	120:
	// Set Parameters to read the Micro Controller (MC1) 3300mv Nominal Voltage INPUT of the EK1914.
		fbCoERead.nSubIndex := 16#01;
		fbCoERead.nIndex 	:= 16#FA81;
		fbCoERead.pDstBuf	:= 	ADR(wEK1914_MC1_3300mV);
		fbCoERead.cbBufLen	:= 	SIZEOF(wEK1914_MC1_3300mV);
		fbCoERead.bExecute	:= TRUE;
		iState := iState + 10;
		
	130:// Evaluate read of the Micro Controller (MC1) 3300mv Nominal Voltage INPUT of the EK1914.		
		IF NOT fbCoERead.bBusy THEN
			q_stEK1914_Diag.lrMC1_3300mV  :=  WORD_TO_LREAL(wEK1914_MC1_3300mV);
			fbCoERead.bExecute	:= FALSE;
			q_sErrorDescription := 'No Error';
			iState := iState + 10;
		ELSIF fbCoERead.bError THEN
			q_sErrorDescription := 'EK1914 MC1 3.3v Input - Read Error';
		END_IF							

	140:
	// Set Parameters to read the Micro Controller (MC2) 3300mv Nominal Voltage INPUT of the EK1914.
		fbCoERead.nSubIndex := 16#02;
		fbCoERead.nIndex 	:= 16#FA81;
		fbCoERead.pDstBuf	:= 	ADR(wEK1914_MC2_3300mV);
		fbCoERead.cbBufLen	:= 	SIZEOF(wEK1914_MC2_3300mV);
		fbCoERead.bExecute	:= TRUE;
		iState := iState + 10;
		
	150:// Evaluate read of the Micro Controller (MC2) 3300mv Nominal Voltage INPUT of the EK1914.		
		IF NOT fbCoERead.bBusy THEN
			q_stEK1914_Diag.lrMC2_3300mV  :=  WORD_TO_LREAL(wEK1914_MC2_3300mV);
			fbCoERead.bExecute	:= FALSE;
			q_sErrorDescription := 'No Error';
			iState := iState + 10;
		ELSIF fbCoERead.bError THEN
			q_sErrorDescription := 'EK1914 MC2 3.3v Input - Read Error';
		END_IF		
	
	160:// Set Parameters to read Standard Output Active/Inactive of the EK1914.
		(* Standard outputs can be used to directly Enable/Disable a TwinSAFE output
	   		if this feature is ACTIVE (Not to Turn it ON/OFF, Allow it or not to turn ON!!! *)
		fbCoERead.nSubIndex := 16#01;
		fbCoERead.nIndex 	:= 16#8000;
		fbCoERead.pDstBuf	:= 	ADR(bEK1914_StandardOuts);
		fbCoERead.cbBufLen	:= 	SIZEOF(bEK1914_StandardOuts);
		fbCoERead.bExecute	:= TRUE;
		iState := iState + 10;
	
	170:// Evaluate read of Standard Output Active/Inactive of the EK1914.
		IF NOT fbCoERead.bBusy THEN								
			q_stEK1914_Diag.xStandardOutputActive  :=  bEK1914_StandardOuts.0 ;
			fbCoERead.bExecute	:= FALSE;
			q_sErrorDescription := 'No Error';
			iState := iState + 10;
		ELSIF fbCoERead.bError THEN
			q_sErrorDescription := 'EK1914 Standard Outputs Active - Read Error';
		END_IF							

	180://Set Parameters to read Test Pulses Active/Inactive of the EK1914.
		(* Used to determine TwinSAFE output wiring is correct *)
		fbCoERead.nSubIndex := 16#03;
		fbCoERead.nIndex 	:= 16#8000;
		fbCoERead.pDstBuf	:= 	ADR(bEK1914_TestP);
		fbCoERead.cbBufLen	:= 	SIZEOF(bEK1914_TestP);
		fbCoERead.bExecute	:= TRUE;
		iState := iState + 10;
		
	190:// Evaluate read of Test Pulses Active/Inactive of the EK1914.
		IF NOT fbCoERead.bBusy THEN								
			q_stEK1914_Diag.xTestPulsesActive  :=  bEK1914_TestP.0 ;
			fbCoERead.bExecute	:= FALSE;
			q_sErrorDescription := 'No Error';
			iState := iState + 10;
		ELSIF fbCoERead.bError THEN
			q_sErrorDescription := 'EK1914 Test Pulses Active/Inactive - Read Error';
		END_IF		

	200:// Set Parameters to read Output Error Acknowledge Active/Inactive of the EK1914.
		(* Used to reset TwinSAFE output errors instead of forcing a cycle power
			for a TwinSAFE output error. *)
		fbCoERead.nSubIndex := 16#04;
		fbCoERead.nIndex 	:= 16#8000;
		fbCoERead.pDstBuf	:= 	ADR(bEK1914_ErrAck);
		fbCoERead.cbBufLen	:= 	SIZEOF(bEK1914_ErrAck);
		fbCoERead.bExecute	:= TRUE;
		iState := iState + 10;
		
	210:// Evaluate read of Output Error Acknowledge Active/Inactive of the EK1914.	
		IF NOT fbCoERead.bBusy THEN								
			q_stEK1914_Diag.xOutputErrAckActive  :=  bEK1914_ErrAck.0 ;
			fbCoERead.bExecute	:= FALSE;
			q_sErrorDescription := 'No Error';
			iState := iState + 10;
		ELSIF fbCoERead.bError THEN
			q_sErrorDescription := 'EK1914 Output Error Acknowledge Active/Inactive - Read Error';
		END_IF						
		
	220:// Set Parameters to read Sensor Tests Active/Inactive Channel 1 of the EK1914.
		fbCoERead.nSubIndex := 1;
		fbCoERead.nIndex 	:= 16#8001;
		fbCoERead.pDstBuf	:= 	ADR(iEK1914_STActive1);
		fbCoERead.cbBufLen	:= 	SIZEOF(iEK1914_STActive1);
		fbCoERead.bExecute	:= TRUE;
		iState := iState + 10;
	
	230:// Evaluate read of	Sensor Tests Active/Inactive Channel 1 of the EK1914.
		IF NOT fbCoERead.bBusy THEN								
			IF NOT iEK1914_STActive1 THEN
				q_stEK1914_Diag.xSensorTestActive1 := FALSE;
			ELSIF iEK1914_STActive1 THEN
				q_stEK1914_Diag.xSensorTestActive1 := TRUE;
			END_IF
			fbCoERead.bExecute	:= FALSE;
			q_sErrorDescription := 'No Error';
			iState := iState + 10;
		ELSIF fbCoERead.bError THEN
			q_sErrorDescription := 'EK1914 Sensor Tests Active/Inactive Channel 1 - Read Error';
		END_IF						
		
	240:// Set Parameters to read Sensor Tests Active/Inactive Channel 2 of the EK1914.
		fbCoERead.nSubIndex := 2;
		fbCoERead.nIndex 	:= 16#8001;
		fbCoERead.pDstBuf	:= 	ADR(iEK1914_STActive2);
		fbCoERead.cbBufLen	:= 	SIZEOF(iEK1914_STActive2);
		fbCoERead.bExecute	:= TRUE;
		iState := iState + 10;
		
	250:// Evaluate read of	Sensor Tests Active/Inactive Channel 1 of the EK1914.
		IF NOT fbCoERead.bBusy THEN								
			IF NOT iEK1914_STActive2 THEN
				q_stEK1914_Diag.xSensorTestActive2 := FALSE;
			ELSIF iEK1914_STActive2 THEN
				q_stEK1914_Diag.xSensorTestActive2 := TRUE;
			END_IF
			fbCoERead.bExecute	:= FALSE;
			q_sErrorDescription := 'No Error';
			iState := iState + 10;
		ELSIF fbCoERead.bError THEN
			q_sErrorDescription := 'EK1914 Sensor Tests Active/Inactive Channel 2 - Read Error';
		END_IF						
		
	260:// Set Parameters to read the Logic setting of Channels 1 and 2 of the EK1914.
		fbCoERead.nSubIndex := 1;
		fbCoERead.nIndex 	:= 16#8002;
		fbCoERead.pDstBuf	:= 	ADR(bEK1914_Logic1_2);
		fbCoERead.cbBufLen	:= 	SIZEOF(bEK1914_Logic1_2);
		fbCoERead.bExecute	:= TRUE;
		iState := iState + 10;
		
	270:// Evaluate read of the Logic setting of Channels 1 and 2 of the EK1914.
		IF NOT fbCoERead.bBusy THEN								
			IF  bEK1914_Logic1_2  = 0  THEN
				q_stEK1914_Diag.sLogicMode_Ch1Ch2 := 'Single Channel Logic.' ;
			ELSIF  bEK1914_Logic1_2  =  1  THEN
				q_stEK1914_Diag.sLogicMode_Ch1Ch2 := 'Asynchronous Repetitive OSSD, Sensor Test Must Be Disabled!' ;
			ELSIF  bEK1914_Logic1_2  =  2  THEN
				q_stEK1914_Diag.sLogicMode_Ch1Ch2 := 'Any Pulse Repetitive OSSD, Sensor Test Must Be Disabled!' ;
			ELSIF  bEK1914_Logic1_2  =  3  THEN
				q_stEK1914_Diag.sLogicMode_Ch1Ch2 := 'Short Cut, No Module Fault.' ;
			ELSE
				q_stEK1914_Diag.sLogicMode_Ch1Ch2 := 'Invalid Logic CH1 and CH2' ;
			END_IF ;		
			fbCoERead.bExecute	:= FALSE;
			q_sErrorDescription := 'No Error';
			iState := iState + 10;
		ELSIF fbCoERead.bError THEN
			q_sErrorDescription := 'EK1914 Logic setting of Channels 1 and 2 - Read Error';
		END_IF						
	
	
(**************************************ALARMS**************************************)
(**************************************ALARMS**************************************)
(**************************************ALARMS**************************************)
	280:// Set Parameters to read the Sensor Test state of the EK1914.	
		fbCoERead.nSubIndex := 16#0A;
		fbCoERead.nIndex 	:= 16#800E;
		fbCoERead.pDstBuf	:= 	ADR(wEK1914_SenT);
		fbCoERead.cbBufLen	:= 	SIZEOF(wEK1914_SenT);
		fbCoERead.bExecute	:= TRUE;
		iState := iState + 10;

	290:// Evaluate read of the Sensor Test state of the EK1914.
		IF NOT fbCoERead.bBusy THEN									
		(* These errors may only be present temporarily so they need to be latched and then cleared
			to be properly noted by the operator. *)
			IF wEK1914_SenT.0 OR wEK1914_SenT.1 THEN
				q_stEK1914_Diag.xSensorTest1_Error 	:= 	wEK1914_SenT.0;
				q_stEK1914_Diag.xSensorTest2_Error 	:= 	wEK1914_SenT.1;
			ELSIF i_xLatchedMessageReset THEN
				q_stEK1914_Diag.xSensorTest1_Error	:= FALSE;
				q_stEK1914_Diag.xSensorTest2_Error	:= FALSE;
			END_IF		
			fbCoERead.bExecute	:= FALSE;
			q_sErrorDescription := 'No Error';
			iState := iState + 10;
		ELSIF fbCoERead.bError THEN
			q_sErrorDescription := 'EK1914 Sensor Test - Read Error';
		END_IF						

	300:// Set Parameters to read the Two-Channel Evaluation Error - Diagnostic object 800E:0B
		(* The two channels contradict each other (not same value). *)
		fbCoERead.nSubIndex := 16#0B;
		fbCoERead.nIndex 	:= 16#800E;
		fbCoERead.pDstBuf	:= 	ADR(wEK1914_2CHEval);
		fbCoERead.cbBufLen	:= 	SIZEOF(wEK1914_2CHEval);
		fbCoERead.bExecute	:= TRUE;
		iState := iState + 10;

	310:// Evalutate read ofthe Two-Channel Evaluation Error - Diagnostic object 800E:0B
		(* The two channels contradict each other (not same value). *)
		IF NOT fbCoERead.bBusy THEN								
		(* These errors may only be present temporarily so they need to be latched and then cleared
			to be properly noted by the operator. *)
			IF wEK1914_2CHEval.0 OR wEK1914_2CHEval.1 THEN
				q_stEK1914_Diag.x2ChanEvalError_Pair1	 :=  wEK1914_2CHEval.0;
			ELSIF i_xLatchedMessageReset THEN
				q_stEK1914_Diag.x2ChanEvalError_Pair1	:= FALSE;
			END_IF	
			fbCoERead.bExecute	:= FALSE;
			q_sErrorDescription := 'No Error';
			iState := iState + 10;
		ELSIF fbCoERead.bError THEN
			q_sErrorDescription := 'EK1914 Two-Channel Evaluation Error - Read Error';
		END_IF						
		
	320:// Set Parameters to read Error In Safety Mat Operating Mode: Input Pair Disagree - Diagnostic object 800E:0C
		(* Input pairs not in the same state (not same value). *)
		fbCoERead.nSubIndex := 16#0C;
		fbCoERead.nIndex 	:= 16#800E;
		fbCoERead.pDstBuf	:= 	ADR(wEK1914_SMiPair);
		fbCoERead.cbBufLen	:= 	SIZEOF(wEK1914_SMiPair);
		fbCoERead.bExecute	:= TRUE;
		iState := iState + 10;
		
	330:// Evaluate read of Error In Safety Mat Operating Mode: Input Pair Disagree - Diagnostic object 800E:0C 
		(* Input pairs not in the same state (not same value). *)
		IF NOT fbCoERead.bBusy THEN								
		(* These errors may only be present temporarily so they need to be latched and then cleared
			to be properly noted by the operator. *)
			IF (wEK1914_SMiPair.0 AND wEK1914_SMiPair.1) THEN
				q_stEK1914_Diag.xSafeMatError_Pair1	 :=  (wEK1914_SMiPair.0  AND  wEK1914_SMiPair.1);
			ELSIF i_xLatchedMessageReset THEN
				q_stEK1914_Diag.xSafeMatError_Pair1	:= FALSE;
			END_IF	
			fbCoERead.bExecute	:= FALSE;
			q_sErrorDescription := 'No Error';
			iState := iState + 10;
		ELSIF fbCoERead.bError THEN
			q_sErrorDescription := 'EK1914 Error In Safety Mat: Input Pair Disagree - Read Error';
		END_IF						
		
	340:// Set Parameters to read Error In Safety Mat Operating Mode: External Supply (No test pulses) - Diagnostic object 800E:0D
		(* External supply detected (Input channel not getting test pulses). *)
		fbCoERead.nSubIndex := 16#0D;
		fbCoERead.nIndex 	:= 16#800E;
		fbCoERead.pDstBuf	:= 	ADR(wEK1914_SMExtSupply);
		fbCoERead.cbBufLen	:= 	SIZEOF(wEK1914_SMExtSupply);
		fbCoERead.bExecute	:= TRUE;
		iState := iState + 10;
		
	350:// Evaluate read Error In Safety Mat Operating Mode: External Supply (No test pulses) - Diagnostic object 800E:0D
		(* External supply detected (Input channel not getting test pulses). *)
		IF NOT fbCoERead.bBusy THEN								
		(* These errors may only be present temporarily so they need to be latched and then cleared
			to be properly noted by the operator. *)
			IF wEK1914_SMExtSupply > 0  THEN
				q_stEK1914_Diag.xSafeMatExternalSupplyErrorCh1  := 	wEK1914_SMExtSupply.0;
				q_stEK1914_Diag.xSafeMatExternalSupplyErrorCh2  := 	wEK1914_SMExtSupply.2;
			ELSIF i_xLatchedMessageReset THEN
				q_stEK1914_Diag.xSafeMatExternalSupplyErrorCh1	:= FALSE;
				q_stEK1914_Diag.xSafeMatExternalSupplyErrorCh2	:= FALSE;
			END_IF
			fbCoERead.bExecute	:= FALSE;
			q_sErrorDescription := 'No Error';
			iState := iState + 10;
		ELSIF fbCoERead.bError THEN
			q_sErrorDescription := 'EK1914 Error In Safety Mat: External Supply - Read Error';
		END_IF						
		
	360:// Set Parameters to read Error At The Output MC1 of the EK1914.
		(* External supply or cross-circuit Error Open Load, Current Below 20mA, OR Current Above Maximum Value OF 500mA. *)
		fbCoERead.nSubIndex := 16#0E;
		fbCoERead.nIndex 	:= 16#800E;
		fbCoERead.pDstBuf	:= 	ADR(wEK1914_OutErrMC1);
		fbCoERead.cbBufLen	:= 	SIZEOF(wEK1914_OutErrMC1);
		fbCoERead.bExecute	:= TRUE;
		iState := iState + 10;
		
	370:// Evaluate read Error At The Output MC1 of the EK1914.
		(* External supply or cross-circuit Error Open Load, Current Below 20mA, OR Current Above Maximum Value OF 500mA. *)	
		IF NOT fbCoERead.bBusy THEN														
		(* These errors may only be present temporarily so they need to be latched and then cleared
			to be properly noted by the operator. *)
			IF wEK1914_OutErrMC1 = 5 THEN
				q_stEK1914_Diag.xCrossCircuitError1_MC1 := TRUE;
				q_stEK1914_Diag.sOutputErrorDescription_MC1 := 'Cross-circuit output 1 and output 2.';
			ELSIF wEK1914_OutErrMC1 = 6 THEN
				q_stEK1914_Diag.xCrossCircuitError2_MC1 := TRUE;
				q_stEK1914_Diag.sOutputErrorDescription_MC1 := 'Cross-circuit output 1 and output 2.';
			ELSIF wEK1914_OutErrMC1 = 10 THEN
				q_stEK1914_Diag.xOverVoltage_MC1 := TRUE;
				q_stEK1914_Diag.sOutputErrorDescription_MC1 := 'Overvoltage.';
			ELSIF wEK1914_OutErrMC1 = 11 THEN
				q_stEK1914_Diag.xUnderVoltage_MC1 := TRUE;
				q_stEK1914_Diag.sOutputErrorDescription_MC1 := 'Undervoltage.';
			ELSIF (wEK1914_OutErrMC1 >= 21) AND (wEK1914_OutErrMC1 <= 27) THEN
				q_stEK1914_Diag.xFieldVoltageError_MC1 := TRUE;
				q_stEK1914_Diag.sOutputErrorDescription_MC1 := 'Error when testing the field voltage switches.';
			ELSIF (wEK1914_OutErrMC1 >= 30) AND (wEK1914_OutErrMC1 <= 33) THEN
				q_stEK1914_Diag.xStartupOutCircuitError_MC1 := TRUE;
				q_stEK1914_Diag.sOutputErrorDescription_MC1 := 'Start-up of the output circuit failed.';
			ELSIF wEK1914_OutErrMC1 = 101 THEN
				q_stEK1914_Diag.xExternalSupply0vError1_MC1 := TRUE;
				q_stEK1914_Diag.sOutputErrorDescription_MC1 := 'External supply 0v output 1, detected with set output.';
			ELSIF wEK1914_OutErrMC1 = 102 THEN
				q_stEK1914_Diag.xExternalSupply24vError1_MC1 := TRUE;
				q_stEK1914_Diag.sOutputErrorDescription_MC1 := 'External supply 24v output 1.';
			ELSIF wEK1914_OutErrMC1 = 103 THEN
				q_stEK1914_Diag.xExternalSupply0vError2_MC1 := TRUE;
				q_stEK1914_Diag.sOutputErrorDescription_MC1 := 'External supply 0v output 2, detected with set output.';
			ELSIF wEK1914_OutErrMC1 = 104 THEN
				q_stEK1914_Diag.xExternalSupply24vError2_MC1 := TRUE;
				q_stEK1914_Diag.sOutputErrorDescription_MC1 := 'External supply 24v output 2.';
			ELSE
				q_stEK1914_Diag.xExternalSupply24vError2_MC1 := FALSE;
				q_stEK1914_Diag.sOutputErrorDescription_MC1 := 'No Error.';
			END_IF
			fbCoERead.bExecute	:= FALSE;
			q_sErrorDescription := 'No Error';
			iState := iState + 10;
		ELSIF fbCoERead.bError THEN
			q_sErrorDescription := 'EK1914 Error At The Output (MC1) - Read Error';
		END_IF		
		
	380:// Set Parameters to read Error At The Output MC2 of the EK1914.
		(* External supply or cross-circuit Error Open Load, Current Below 20mA, OR Current Above Maximum Value OF 500mA. *)
		fbCoERead.nSubIndex := 16#0F;
		fbCoERead.nIndex 	:= 16#800E;
		fbCoERead.pDstBuf	:= 	ADR(wEK1914_OutErrMC2);
		fbCoERead.cbBufLen	:= 	SIZEOF(wEK1914_OutErrMC2);
		fbCoERead.bExecute	:= TRUE;
		iState := iState + 10;
	
	390:// Evaluate read of Error At The Output MC2 of the EK1914.
		(* External supply or cross-circuit Error Open Load, Current Below 20mA, OR Current Above Maximum Value OF 500mA. *)
		IF NOT fbCoERead.bBusy THEN	
		(* These errors may only be present temporarily so they need to be latched and then cleared
			to be properly noted by the operator. *)
			IF wEK1914_OutErrMC2 = 5 THEN
				q_stEK1914_Diag.xCrossCircuitError1_MC2 := TRUE;
				q_stEK1914_Diag.sOutputErrorDescription_MC2 := 'Cross-circuit output 1 and output 2 MC2.';
			ELSIF wEK1914_OutErrMC2 = 6 THEN
				q_stEK1914_Diag.xCrossCircuitError2_MC2 := TRUE;
				q_stEK1914_Diag.sOutputErrorDescription_MC2 := 'Cross-circuit output 1 and output 2 MC2.';
			ELSIF wEK1914_OutErrMC2 = 10 THEN
				q_stEK1914_Diag.xOverVoltage_MC2 := TRUE;
				q_stEK1914_Diag.sOutputErrorDescription_MC2 := 'Overvoltage MC2.';
			ELSIF wEK1914_OutErrMC2 = 11 THEN
				q_stEK1914_Diag.xUnderVoltage_MC2 := TRUE;
				q_stEK1914_Diag.sOutputErrorDescription_MC2 := 'Undervoltage.';
			ELSIF (wEK1914_OutErrMC2 >= 21) AND (wEK1914_OutErrMC2 <= 27) THEN
				q_stEK1914_Diag.xFieldVoltageError_MC2 := TRUE;
				q_stEK1914_Diag.sOutputErrorDescription_MC2 := 'Error when testing the field voltage switches MC2.';
			ELSIF (wEK1914_OutErrMC2 >= 30) AND (wEK1914_OutErrMC2 <= 33) THEN
				q_stEK1914_Diag.xStartupOutCircuitError_MC2 := TRUE;
				q_stEK1914_Diag.sOutputErrorDescription_MC2 := 'Start-up of the output circuit failed MC2.';
			ELSIF wEK1914_OutErrMC2 = 101 THEN
				q_stEK1914_Diag.xExternalSupply0vError1_MC2 := TRUE;
				q_stEK1914_Diag.sOutputErrorDescription_MC2 := 'External supply 0v output 1, detected with set output MC2.';
			ELSIF wEK1914_OutErrMC2 = 102 THEN
				q_stEK1914_Diag.xExternalSupply24vError1_MC2 := TRUE;
				q_stEK1914_Diag.sOutputErrorDescription_MC2 := 'External supply 24v output 1 MC2.';
			ELSIF wEK1914_OutErrMC2 = 103 THEN
				q_stEK1914_Diag.xExternalSupply0vError2_MC2 := TRUE;
				q_stEK1914_Diag.sOutputErrorDescription_MC2 := 'External supply 0v output 2, detected with set output MC2.';
			ELSIF wEK1914_OutErrMC2 = 104 THEN
				q_stEK1914_Diag.xExternalSupply24vError2_MC2 := TRUE;
				q_stEK1914_Diag.sOutputErrorDescription_MC2 := 'External supply 24v output 2 MC2.';
			ELSE
				q_stEK1914_Diag.xExternalSupply24vError2_MC2 := FALSE;
				q_stEK1914_Diag.sOutputErrorDescription_MC2 := 'No Error.';
			END_IF
			fbCoERead.bExecute	:= FALSE;
			q_sErrorDescription := 'No Error';
			iState := iState + 10;
		ELSIF fbCoERead.bError THEN
			q_sErrorDescription := 'EK1914 Error At The Output (MC2) - Read Error';
		END_IF								

	400:// Set Parameters to read Connection State of the EK1914.
		fbCoERead.nSubIndex := 1;
		fbCoERead.nIndex 	:= 16#A000;
		fbCoERead.pDstBuf	:= 	ADR(iEK1914_ConnectionState);
		fbCoERead.cbBufLen	:= 	SIZEOF(iEK1914_ConnectionState);
		fbCoERead.bExecute	:= TRUE;
		iState := iState + 10;
		
	410:// Evaluate read of the Connection State of the EK1914.
		IF NOT fbCoERead.bBusy THEN								
			IF iEK1914_ConnectionState = 100 THEN
				q_stEK1914_Diag.sConnectionState := 'Reset State';
			ELSIF iEK1914_ConnectionState = 101 THEN
				q_stEK1914_Diag.sConnectionState := 'Session State';
			ELSIF iEK1914_ConnectionState = 102 THEN
				q_stEK1914_Diag.sConnectionState := 'Connection State';
			ELSIF iEK1914_ConnectionState = 103 THEN
				q_stEK1914_Diag.sConnectionState := 'Parameter State';
			ELSIF iEK1914_ConnectionState = 104 THEN
				q_stEK1914_Diag.sConnectionState := 'Data State';
			ELSIF iEK1914_ConnectionState = 105 THEN
				q_stEK1914_Diag.sConnectionState := 'Failsafe State';
			ELSE
				q_stEK1914_Diag.sConnectionState := 'Undefined State';
			END_IF
			fbCoERead.bExecute	:= FALSE;
			q_sErrorDescription := 'No Error';
			iState := 0;
		ELSIF fbCoERead.bError THEN
			q_sErrorDescription := 'EK1914 Connection State - Read Error';
		END_IF	
END_CASE

// FB_EcCoESdoRead for all CoE reads.
fbCoERead(
	sNetId:= i_sNetId, 
	nSlaveAddr:= i_nSlaveAddr, 
	nSubIndex:= , 
	nIndex:= , 
	pDstBuf:= , 
	cbBufLen:= , 
	bExecute:= , 
	tTimeout:= T#2S, 
	bBusy=> , 
	bError=> q_xError, 
	nErrId=> q_udiErrorID);

// If any of above errors exist set q_stEK1914_Diag.xEK1914Error TRUE.
IF NOT q_stEK1914_Diag.xSensorTest1_Error OR
		q_stEK1914_Diag.xSensorTest2_Error OR
		q_stEK1914_Diag.x2ChanEvalError_Pair1 OR
		q_stEK1914_Diag.xSafeMatError_Pair1 OR
		q_stEK1914_Diag.xSafeMatExternalSupplyErrorCh1 OR
		q_stEK1914_Diag.xSafeMatExternalSupplyErrorCh2 OR 
		q_stEK1914_Diag.xCrossCircuitError1_MC1 OR 
		q_stEK1914_Diag.xCrossCircuitError2_MC1 OR 
		q_stEK1914_Diag.xOverVoltage_MC1 OR 
		q_stEK1914_Diag.xUnderVoltage_MC1 OR
		q_stEK1914_Diag.xFieldVoltageError_MC1 OR 
		q_stEK1914_Diag.xStartupOutCircuitError_MC1 OR 
		q_stEK1914_Diag.xExternalSupply0vError1_MC1 OR 
		q_stEK1914_Diag.xExternalSupply24vError1_MC1 OR 
		q_stEK1914_Diag.xExternalSupply0vError2_MC1 OR 
		q_stEK1914_Diag.xExternalSupply24vError2_MC1 OR
		q_stEK1914_Diag.xCrossCircuitError1_MC2 OR 
		q_stEK1914_Diag.xCrossCircuitError2_MC2 OR 
		q_stEK1914_Diag.xOverVoltage_MC2 OR 
		q_stEK1914_Diag.xUnderVoltage_MC2 OR
		q_stEK1914_Diag.xFieldVoltageError_MC2 OR 
		q_stEK1914_Diag.xStartupOutCircuitError_MC2 OR 
		q_stEK1914_Diag.xExternalSupply0vError1_MC2 OR 
		q_stEK1914_Diag.xExternalSupply24vError1_MC2 OR 
		q_stEK1914_Diag.xExternalSupply0vError2_MC2 OR 
		q_stEK1914_Diag.xExternalSupply24vError2_MC2 THEN
			q_stEK1914_Diag.xEK1914Error := FALSE;
ELSIF q_stEK1914_Diag.xSensorTest1_Error OR
		q_stEK1914_Diag.xSensorTest2_Error OR
		q_stEK1914_Diag.x2ChanEvalError_Pair1 OR
		q_stEK1914_Diag.xSafeMatError_Pair1 OR
		q_stEK1914_Diag.xSafeMatExternalSupplyErrorCh1 OR
		q_stEK1914_Diag.xSafeMatExternalSupplyErrorCh2 OR 
		q_stEK1914_Diag.xCrossCircuitError1_MC1 OR 
		q_stEK1914_Diag.xCrossCircuitError2_MC1 OR 
		q_stEK1914_Diag.xOverVoltage_MC1 OR 
		q_stEK1914_Diag.xUnderVoltage_MC1 OR
		q_stEK1914_Diag.xFieldVoltageError_MC1 OR 
		q_stEK1914_Diag.xStartupOutCircuitError_MC1 OR 
		q_stEK1914_Diag.xExternalSupply0vError1_MC1 OR 
		q_stEK1914_Diag.xExternalSupply24vError1_MC1 OR 
		q_stEK1914_Diag.xExternalSupply0vError2_MC1 OR 
		q_stEK1914_Diag.xExternalSupply24vError2_MC1 OR
		q_stEK1914_Diag.xCrossCircuitError1_MC2 OR 
		q_stEK1914_Diag.xCrossCircuitError2_MC2 OR 
		q_stEK1914_Diag.xOverVoltage_MC2 OR 
		q_stEK1914_Diag.xUnderVoltage_MC2 OR
		q_stEK1914_Diag.xFieldVoltageError_MC2 OR 
		q_stEK1914_Diag.xStartupOutCircuitError_MC2 OR 
		q_stEK1914_Diag.xExternalSupply0vError1_MC2 OR 
		q_stEK1914_Diag.xExternalSupply24vError1_MC2 OR 
		q_stEK1914_Diag.xExternalSupply0vError2_MC2 OR 
		q_stEK1914_Diag.xExternalSupply24vError2_MC2 THEN
			q_stEK1914_Diag.xEK1914Error := TRUE;
END_IF

END_FUNCTION_BLOCK

// POUs/HardwareFBs/FB_EL69xxDiagnostics
(*=====================================================================
Beckhoff Automation LLC
Copyright 2015 All Rights Reserved
=======================================================================
Description: 
This Program has been supplied by Beckhoff Automation As-Is and is intended only as an example implementation. 
Functionality is not guaranteed. 
This Function Block reads all status and error information known at time of creation of the EL69xx.
---------------------------------------------------------------------------------------------------------------
History:
Date		Version			Author							Comment
---------------------------------------------------------------------------------------------------------------
07.08.15	0.10		Jason Erickson				Initial Library Creation.
07.20.15	0.11		Jason Ericskon				Added CoE Read for TwinSAFE Connection State.
08.28.15	0.20		Jason Erickson				Code optimization to eliminate timed data reads.
09.18.15	0.2.1		Jason Erickson				Added new error codes 0x6000 - 0x6002 and Connection Status to the AX5805.
09.24.15	0.2.2		Jason Erickson				Corrected inability to update CASE in FB_EL1904Diagnostics and FB_EL2904Diagnostics.
10.30.15	0.2.3		Jason Erickson				Modified Diagnostic Structure names for ease of use.
*)
FUNCTION_BLOCK FB_EL69xxDiagnostics
VAR_INPUT
// EtherCAT Master Device Net ID.
	i_sNetId: STRING;
// Slave Address of the EL69xx.
	i_nSlaveAddr: UINT;
// Input to reset Latched TwinSAFE Error Messages.
	i_xLatchedMessageReset: BOOL;
END_VAR
VAR_OUTPUT
// Structure to hold all EL69xx output information.
	q_stEL69xx_Diag: ST_EL69xx_DIAGNOSTICS;
// Internal function block errors.
	q_xError: BOOL;
	q_udiErrorID: UDINT;
	q_sErrorDescription: STRING;
END_VAR
VAR
// Case Statement.
	iState: INT;
// FB_EcCoESdoRead for all CoE reads.
	fbCoERead: FB_EcCoESdoRead;
// Variable to hold data for evaluation, Micro Controller (MC1) 3.3v Nominal Voltage(mV) INPUT of the EL69xx.
	wEL69xx_MC1_3300mV: WORD;
// Variable to hold data for evaluation, Micro Controller (MC2) 3.3v Nominal Voltage(mV) INPUT of the EL69xx.
	wEL69xx_MC2_3300mV: WORD;
// Variable to hold data for evaluation, Temperature and Voltage Errors of the EL69xx.
	(* There are two temperature sensors inside each Microcontroller. *)
	wEL69xx_Error: WORD;
END_VAR

CASE iState OF
	0:
	// Set Parameters to read Serial Number of the EL69xx.	
		fbCoERead.nSubIndex := 16#02;
		fbCoERead.nIndex 	:= 16#F980;
		fbCoERead.pDstBuf	:= 	ADR(q_stEL69xx_Diag.dwSerialNumber);
		fbCoERead.cbBufLen	:= 	SIZEOF(q_stEL69xx_Diag.dwSerialNumber);
		fbCoERead.bExecute	:= TRUE;
		iState := iState + 10;
		
	10:// Evaluate read of the Serial Number of the EL69xx.
		IF NOT fbCoERead.bBusy THEN
			fbCoERead.bExecute	:= FALSE;
			q_sErrorDescription := 'No Error';
			iState := iState + 10;
		ELSIF fbCoERead.bError THEN
			q_sErrorDescription := 'EL69xx Serial Number - Read Error';
		END_IF
	
	20:// Set Parameters to read DIP Switch setting out of the EL69xx.
		fbCoERead.nSubIndex := 16#01;
		fbCoERead.nIndex 	:= 16#F980;
		fbCoERead.pDstBuf	:= 	ADR(q_stEL69xx_Diag.wDipSwitch);
		fbCoERead.cbBufLen	:= 	SIZEOF(q_stEL69xx_Diag.wDipSwitch);
		fbCoERead.bExecute	:= TRUE;
		iState := iState + 10;
		
	30:// Evaluate read of the DIP Switch setting of the EL69xx.
		IF NOT fbCoERead.bBusy THEN
			fbCoERead.bExecute	:= FALSE;
			q_sErrorDescription := 'No Error';
			iState := iState + 10;
		ELSIF fbCoERead.bError THEN
			q_sErrorDescription := 'EL69xx DIP Switch - Read Error';
		END_IF	
	
	40:// Set Parameters to read Hardware Version of the EL69xx.
		fbCoERead.nSubIndex := 0;
		fbCoERead.nIndex 	:= 16#1009;
		fbCoERead.pDstBuf	:= 	ADR(q_stEL69xx_Diag.sHwVersion);
		fbCoERead.cbBufLen	:= 	SIZEOF(q_stEL69xx_Diag.sHwVersion);
		fbCoERead.bExecute	:= TRUE;
		iState := iState + 10;
	
	50:// Evaluate read of Hardware Version of the EL69xx.
		IF NOT fbCoERead.bBusy THEN
			fbCoERead.bExecute	:= FALSE;
			q_sErrorDescription := 'No Error';
			iState := iState + 10;
		ELSIF fbCoERead.bError THEN
			q_sErrorDescription := 'EL69xx Hardware Version - Read Error';
		END_IF	

	60:// Set Parameters to read Software Version (firmware) of the EL69xx.
		fbCoERead.nSubIndex := 0;
		fbCoERead.nIndex 	:= 16#100A;
		fbCoERead.pDstBuf	:= 	ADR(q_stEL69xx_Diag.sFwVersion);
		fbCoERead.cbBufLen	:= 	SIZEOF(q_stEL69xx_Diag.sFwVersion);
		fbCoERead.bExecute	:= TRUE;
		iState := iState + 10;
	
	70:// Evaluate read of Software Version (firmware) of the EL69xx.
		IF NOT fbCoERead.bBusy THEN
			fbCoERead.bExecute	:= FALSE;
			q_sErrorDescription := 'No Error';
			iState := iState + 10;
		ELSIF fbCoERead.bError THEN
			q_sErrorDescription := 'EL69xx Software Version - Read Error';
		END_IF	

	80:// Set Parameters to read Micro Controller (MC1) Temperature in DegC of the EL69xx.
		fbCoERead.nSubIndex := 1;
		fbCoERead.nIndex 	:= 16#FA80;
		fbCoERead.pDstBuf	:= 	ADR(q_stEL69xx_Diag.wMC1Temp);
		fbCoERead.cbBufLen	:= 	SIZEOF(q_stEL69xx_Diag.wMC1Temp);
		fbCoERead.bExecute	:= TRUE;
		iState := iState + 10;
		
	90:// Evaluate read of Micro Controller (MC1) Temperature in DegC of the EL69xx.
		IF NOT fbCoERead.bBusy THEN
			fbCoERead.bExecute	:= FALSE;
			q_sErrorDescription := 'No Error';
			iState := iState + 10;
		ELSIF fbCoERead.bError THEN
			q_sErrorDescription := 'EL69xx MC1 Temp - Read Error';
		END_IF

	100:// Set Parameters to read Micro Controller (MC2) Temperature in DegC of the EL69xx.
		fbCoERead.nSubIndex := 2;
		fbCoERead.nIndex 	:= 16#FA80;
		fbCoERead.pDstBuf	:= 	ADR(q_stEL69xx_Diag.wMC2Temp);
		fbCoERead.cbBufLen	:= 	SIZEOF(q_stEL69xx_Diag.wMC2Temp);
		fbCoERead.bExecute	:= TRUE;
		iState := iState + 10;
		
	110:// Evaluate read of Micro Controller (MC2) Temperature in DegC of the EL69xx.
		IF NOT fbCoERead.bBusy THEN
			fbCoERead.bExecute	:= FALSE;
			q_sErrorDescription := 'No Error';
			iState := iState + 10;
		ELSIF fbCoERead.bError THEN
			q_sErrorDescription := 'EL69xx MC2 Temp - Read Error';
		END_IF

	120://Set Parameters to read Micro Controller (MC1) 3300mv Nominal Voltage INPUT of the EL69xx.
		fbCoERead.nSubIndex := 3;
		fbCoERead.nIndex 	:= 16#FA80;
		fbCoERead.pDstBuf	:= 	ADR(wEL69xx_MC1_3300mV);
		fbCoERead.cbBufLen	:= 	SIZEOF(wEL69xx_MC1_3300mV);
		fbCoERead.bExecute	:= TRUE;
		iState := iState + 10;
		
	130:// Evaluate read of Micro Controller (MC1) 3300mv Nominal Voltage INPUT of the EL69xx.
		IF NOT fbCoERead.bBusy THEN
			q_stEL69xx_Diag.lrMC1_3300mV  :=  WORD_TO_LREAL(wEL69xx_MC1_3300mV);
			fbCoERead.bExecute	:= FALSE;
			q_sErrorDescription := 'No Error';
			iState := iState + 10;
		ELSIF fbCoERead.bError THEN
			q_sErrorDescription := 'EL69xx MC1 3.3v Input - Read Error';
		END_IF

	140:// Set Parameters to read Micro Controller (MC2) 3300mv Nominal Voltage INPUT of the EL69xx.
		fbCoERead.nSubIndex := 4;
		fbCoERead.nIndex 	:= 16#FA80;
		fbCoERead.pDstBuf	:= 	ADR(wEL69xx_MC2_3300mV);
		fbCoERead.cbBufLen	:= 	SIZEOF(wEL69xx_MC2_3300mV);
		fbCoERead.bExecute	:= TRUE;
		iState := iState + 10;
		
	150:// Evaluate read of	Micro Controller (MC2) 3300mv Nominal Voltage INPUT of the EL69xx.
		IF NOT fbCoERead.bBusy THEN
			q_stEL69xx_Diag.lrMC2_3300mV  :=  WORD_TO_LREAL(wEL69xx_MC2_3300mV);
			fbCoERead.bExecute	:= FALSE;
			q_sErrorDescription := 'No Error';
			iState := iState + 10;
		ELSIF fbCoERead.bError THEN
			q_sErrorDescription := 'EL69xx MC2 3.3v Input Read - Error';
		END_IF
		
	160:// Set Parameters to read Temperature and Voltage Errors of the EL69xx.
		(* There are two temperature sensors inside each Microcontroller. *)
		fbCoERead.nSubIndex := 3;
		fbCoERead.nIndex 	:= 16#FA00;
		fbCoERead.pDstBuf	:= 	ADR(wEL69xx_Error);
		fbCoERead.cbBufLen	:= 	SIZEOF(wEL69xx_Error);
		fbCoERead.bExecute	:= TRUE;
		iState := iState + 10;
	
	170:// Evaluate read of	Temperature and Voltage Errors of the EL69xx.	
		(* There are two temperature sensors inside each Microcontroller. *)
		IF NOT fbCoERead.bBusy THEN
		(* These errors may only be present temporarily so they need to be latched and then cleared
			to be properly noted by the operator. *)
			IF wEL69xx_Error.2 OR wEL69xx_Error.8 THEN
				q_stEL69xx_Diag.xMaxTempError		:= 		(wEL69xx_Error = 5);
				q_stEL69xx_Diag.xMinTempError		:= 		(wEL69xx_Error = 6);
				q_stEL69xx_Diag.xTempDiffError	:= 		(wEL69xx_Error = 7);
				q_stEL69xx_Diag.xMaxVccMC1		:= 		(wEL69xx_Error = 257);
				q_stEL69xx_Diag.xMaxVccMC2		:= 		(wEL69xx_Error = 258);
				q_stEL69xx_Diag.xMinVccMC1		:= 		(wEL69xx_Error = 259);
				q_stEL69xx_Diag.xMinVccMC2		:= 		(wEL69xx_Error = 260);
			ELSIF i_xLatchedMessageReset THEN
				q_stEL69xx_Diag.xMaxTempError	:= FALSE;
				q_stEL69xx_Diag.xMinTempError	:= FALSE;
				q_stEL69xx_Diag.xTempDiffError:= FALSE;
				q_stEL69xx_Diag.xMaxVccMC1	:= FALSE;
				q_stEL69xx_Diag.xMaxVccMC2	:= FALSE;
				q_stEL69xx_Diag.xMinVccMC1	:= FALSE;
				q_stEL69xx_Diag.xMinVccMC2	:= FALSE;
			END_IF
			fbCoERead.bExecute	:= FALSE;
			q_sErrorDescription := 'No Error';
			iState := iState + 10;
		ELSIF fbCoERead.bError THEN
			q_sErrorDescription := 'EL69xx Temp and Voltage Error - Read Error';
		END_IF
		
	180:// Set Parameters to read Number of Safety Connections configured In The EL69xx.
		fbCoERead.nSubIndex := 0;
		fbCoERead.nIndex 	:= 16#2110;
		fbCoERead.pDstBuf	:= 	ADR(q_stEL69xx_Diag.bNumOfConnections);
		fbCoERead.cbBufLen	:= 	SIZEOF(q_stEL69xx_Diag.bNumOfConnections);
		fbCoERead.bExecute	:= TRUE;
		iState := iState + 10;
		
	190:// Evaluate read of Number of Safety Connections configured In The EL69xx.
		IF NOT fbCoERead.bBusy THEN
			fbCoERead.bExecute	:= FALSE;
			q_sErrorDescription := 'No Error';
			iState := iState + 10;
		ELSIF fbCoERead.bError THEN
			q_sErrorDescription := 'EL69xx Number of Safety Connections - Read Error';
		END_IF	

	200:// Set Parameters to read Number of Safety Groups Configured in the EL69xx.
		fbCoERead.nSubIndex := 0;
		fbCoERead.nIndex 	:= 16#2120;
		fbCoERead.pDstBuf	:= 	ADR(q_stEL69xx_Diag.bNumOfSafetyGroups);
		fbCoERead.cbBufLen	:= 	SIZEOF(q_stEL69xx_Diag.bNumOfSafetyGroups);
		fbCoERead.bExecute	:= TRUE;
		iState := iState + 10;
		
	210:// Evaluate read of Number of Safety Groups Configured in the EL69xx.	
		IF NOT fbCoERead.bBusy THEN
			fbCoERead.bExecute	:= FALSE;
			q_sErrorDescription := 'No Error';
			iState := iState + 10;
		ELSIF fbCoERead.bError THEN
			q_sErrorDescription := 'EL69xx Number of Safety Groups - Read Error';
		END_IF	
	
	220://Set Parameters to read Number of Safety Function Blocks Configured in the EL69xx.
		fbCoERead.nSubIndex := 0;
		fbCoERead.nIndex 	:= 16#2130;
		fbCoERead.pDstBuf	:= 	ADR(q_stEL69xx_Diag.bNumOfSafetyBlocks);
		fbCoERead.cbBufLen	:= 	SIZEOF(q_stEL69xx_Diag.bNumOfSafetyBlocks);
		fbCoERead.bExecute	:= TRUE;
		iState := iState + 10;
		
	230:// Evaluate read of	Number of Safety Function Blocks Configured in the EL69xx.
		IF NOT fbCoERead.bBusy THEN
			fbCoERead.bExecute	:= FALSE;
			q_sErrorDescription := 'No Error';
			iState := 0;
		ELSIF fbCoERead.bError THEN
			q_sErrorDescription := 'EL69xx Number of Safety Function Blocks Configured - Read Error';
		END_IF	
END_CASE

// FB_EcCoESdoRead for all CoE reads.
fbCoERead(
	sNetId:= i_sNetId, 
	nSlaveAddr:= i_nSlaveAddr, 
	nSubIndex:= , 
	nIndex:= , 
	pDstBuf:= , 
	cbBufLen:= , 
	bExecute:= , 
	tTimeout:= T#2S, 
	bBusy=> , 
	bError=> q_xError, 
	nErrId=> q_udiErrorID);

// If any of above errors exist set q_stEL69xx_Diag.xEL69xq_xError TRUE
IF NOT q_stEL69xx_Diag.xMaxTempError OR
	q_stEL69xx_Diag.xMinTempError OR
	q_stEL69xx_Diag.xMaxVccMC1 OR
	q_stEL69xx_Diag.xMaxVccMC2 OR
	q_stEL69xx_Diag.xMinVccMC1 OR
	q_stEL69xx_Diag.xMinVccMC2 OR
	q_stEL69xx_Diag.xTempDiffError THEN
		q_stEL69xx_Diag.xEL69xxError := FALSE;
ELSIF q_stEL69xx_Diag.xMaxTempError OR
	q_stEL69xx_Diag.xMinTempError OR
	q_stEL69xx_Diag.xMaxVccMC1 OR
	q_stEL69xx_Diag.xMaxVccMC2 OR
	q_stEL69xx_Diag.xMinVccMC1 OR
	q_stEL69xx_Diag.xMinVccMC2 OR
	q_stEL69xx_Diag.xTempDiffError THEN
		q_stEL69xx_Diag.xEL69xxError := TRUE;
END_IF

END_FUNCTION_BLOCK

// POUs/HardwareFBs/FB_EP1908Diagnostics
(*=====================================================================
Beckhoff Automation LLC
Copyright 2015 All Rights Reserved
=======================================================================
Description: 
This Program has been supplied by Beckhoff Automation As-Is and is intended only as an example implementation. 
Functionality is not guaranteed. 
This Function Block reads all status and error information known at time of creation of the EP1908.
---------------------------------------------------------------------------------------------------------------
History:
Date		Version			Author							Comment
---------------------------------------------------------------------------------------------------------------
07.08.15	0.10		Jason Erickson				Initial Library Creation.
07.20.15	0.11		Jason Ericskon				Added CoE Read for TwinSAFE Connection State.
08.28.15	0.20		Jason Erickson				Code optimization to eliminate timed data reads.
09.18.15	0.2.1		Jason Erickson				Added new error codes 0x6000 - 0x6002 and Connection Status to the AX5805.
09.24.15	0.2.2		Jason Erickson				Corrected inability to update CASE in FB_EL1904Diagnostics and FB_EL2904Diagnostics.
10.30.15	0.2.3		Jason Erickson				Modified Diagnostic Structure names for ease of use.
*)
FUNCTION_BLOCK FB_EP1908Diagnostics
VAR_INPUT
// EtherCAT Master Device Net ID.
	i_sNetId: STRING;
// Slave Address of the EP1908.		
	i_nSlaveAddr: UINT;
// Input to reset Latched TwinSAFE Error Messages.
	i_xLatchedMessageReset: BOOL;
END_VAR
VAR_OUTPUT
// Structure to hold all EP1908 output information.
	q_stEP1908_Diag: ST_EP1908_DIAGNOSTICS;
// Internal function block errors.
	q_xError: BOOL;
	q_nErrorID: UDINT;
	q_sErrorDescription: STRING;
END_VAR
VAR
// Case Statement.
	iState: INT;
// FB_EcCoESdoRead for all CoE reads.
	fbCoERead: FB_EcCoESdoRead;
// FB_EcCoESdoReadEx for all CoE EX reads.
	fbCoEReadEX: FB_EcCoESdoReadEx;
// Variable to hold data for evaluation, Micro Controller (MC1) 3.3v Nominal Voltage(mV) INPUT of the EP1908.	
	wEP1908_MC1_3300mV: WORD;
// Variable to hold data for evaluation, Micro Controller (MC2) 3.3v Nominal Voltage(mV) INPUT of the EP1908.	
	wEP1908_MC2_3300mV: WORD;
// Variable to hold data for evaluation, Operating Mode of the EP1908.
	wEP1908_OperMode: WORD;
// Variable to hold data for evaluation, Sensor Tests Active/Inactive of the EP1908.
	iSensorTestActive: INT;
// Variable to hold data for evaluation, Logic of the EP1908 Channels 1 and 2.
	bEP1908_Logic1_2: BYTE;
// Variable to hold data for evaluation, Logic of the EP1908 Channels 3 and 4.
	bEP1908_Logic3_4: BYTE;
// Variable to hold data for evaluation, Logic of the EP1908 Channels 5 and 6.
	bEP1908_Logic5_6: BYTE;
// Variable to hold data for evaluation, Logic of the EP1908 Channels 7 and 8.
	bEP1908_Logic7_8: BYTE;
// Variable to hold data for evaluation, Velocity/Frequency Limits.
	arrEP1908_VelocityLimit: ARRAY[0..8] OF INT;
// Variable to hold data for evaluation, Actual Velocity/Frequencies.
	arrEP1908ActualVelocities: ARRAY[0..7] OF INT;
// Variable to hold data for evaluation, Max Velocity/Frequencies.
		(* Max value since the last Startup of TwinSAFE. *)
	arrEP1908MaxVelocities: ARRAY[0..7] OF INT;
// Variable to hold data for evaluation, Sensor Test Errors of the EP1908.
	wEP1908_SenT: WORD;
// Variable to hold data for evaluation, Two-Channel Evaluation error of the EP1908.
	wEP1908_2CHEval: WORD;
// Variable to hold data for evaluation, Error In Safety Mat Operating Mode: Input Pair Disagree - Diagnostic object 800E:0C of the EP1908.
		(* The two channels contradict each other (not same value). *)	
	wEP1908_SMiPair: WORD;
// Variable to hold data for evaluation, Error In Safety Mat Operating Mode: External Supply (No test pulses) - Diagnostic object 800E:0D of the EP1908.	
		(* External supply detected (Input channel not getting test pulses). *)	
	wEP1908_SMExtSupply: WORD;
// Variable to hold data for evaluation, Speed Monitoring Error: Overspeed. 
		(* (Overspeed was detected at the input. *)
	wEP1908_SpeedMonitor: WORD;
// Variable to hold data for evaluation, Two Channel Sync Velocity Control Error of the EP1908. 
		(* Both inputs of an input pair were read with inactive State *)
	wEP1908_2ChSyncVelo: WORD;
// Variable to hold data for evaluation, Two Channel Sync Velocity Control AND Two Channel Encoder Velocity Control Error of the EP1908. 
		(* Different speeds were identified for the two inputs of an input pair. *)
	wEP1908_2ChSyncVeloAnd2ChEncVelo: WORD;
	// Variable to hold data for evaluation, Connection State of the EP1908.
	iEP1908_ConnectionState: INT;
END_VAR

CASE iState OF
	0:// Set Parameters to read the Serial Number of the EP1908.			
			fbCoERead.nSubIndex	:= 	16#02;
			fbCoERead.nIndex	:= 	16#F980;
			fbCoERead.pDstBuf	:= 	ADR(q_stEP1908_Diag.dwSerialNumber);
			fbCoERead.cbBufLen	:= 	SIZEOF(q_stEP1908_Diag.dwSerialNumber);
			fbCoERead.bExecute	:= 	TRUE;		
			iState := iState + 10;							
	
	10:// Evaluate read of the Serial Number of the EP1908.			
		IF NOT fbCoERead.bBusy THEN
			fbCoERead.bExecute := FALSE;
			q_sErrorDescription := 'No Error';
			iState := iState + 10;
			IF fbCoERead.bError THEN
				q_sErrorDescription := 'EP1908 Serial Number - Read Error';
			END_IF
		END_IF
	
	20:// Set Parameters to read the DIP Switch setting of the EP1908.			
			fbCoERead.nSubIndex	:= 	16#01;
			fbCoERead.nIndex	:= 	16#F980;
			fbCoERead.pDstBuf	:= 	ADR(q_stEP1908_Diag.wDipSwitch);
			fbCoERead.cbBufLen	:= 	SIZEOF(q_stEP1908_Diag.wDipSwitch);
			fbCoERead.bExecute	:= 	TRUE;		
			iState := iState + 10;							
	
	30:// Evaluate read of the DIP Switch setting of the EP1908.			
		IF NOT fbCoERead.bBusy THEN
			fbCoERead.bExecute := FALSE;
			q_sErrorDescription := 'No Error';
			iState := iState + 10;
			IF fbCoERead.bError THEN
				q_sErrorDescription := 'EP1908 DIP Switch Setting - Read Error';
			END_IF
		END_IF

	40:// Set Parameters to read the Hardware Version of the EP1908.			
			fbCoERead.nSubIndex	:= 	0;
			fbCoERead.nIndex	:= 	16#1009;
			fbCoERead.pDstBuf	:= 	ADR(q_stEP1908_Diag.sHwVersion);
			fbCoERead.cbBufLen	:= 	SIZEOF(q_stEP1908_Diag.sHwVersion);
			fbCoERead.bExecute	:= 	TRUE;		
			iState := iState + 10;							
	
	50:// Evaluate read of the Hardware Version of the EP1908.			
		IF NOT fbCoERead.bBusy THEN
			fbCoERead.bExecute := FALSE;
			q_sErrorDescription := 'No Error';
			iState := iState + 10;
			IF fbCoERead.bError THEN
				q_sErrorDescription := 'EP1908 Hardware Version - Read Error';
			END_IF
		END_IF

	60:// Set Parameters to read the Software Version (firmware) of the EP1908.			
			fbCoERead.nSubIndex	:= 	0;
			fbCoERead.nIndex	:= 	16#100A;
			fbCoERead.pDstBuf	:= 	ADR(q_stEP1908_Diag.sFwVersion);
			fbCoERead.cbBufLen	:= 	SIZEOF(q_stEP1908_Diag.sFwVersion);
			fbCoERead.bExecute	:= 	TRUE;		
			iState := iState + 10;							
	
	70:// Evaluate read of the Software Version (firmware) of the EP1908.			
		IF NOT fbCoERead.bBusy THEN
			fbCoERead.bExecute := FALSE;
			q_sErrorDescription := 'No Error';
			iState := iState + 10;
			IF fbCoERead.bError THEN
				q_sErrorDescription := 'EP1908 Software Version (firmware) - Read Error';
			END_IF
		END_IF
	
	80:// Set Parameters to read Micro Controller (MC1) Temperature in DegC of the EP1908.			
			fbCoERead.nSubIndex	:= 	16#01;
			fbCoERead.nIndex	:= 	16#FA80;
			fbCoERead.pDstBuf	:= 	ADR(q_stEP1908_Diag.wMC1Temp);
			fbCoERead.cbBufLen	:= 	SIZEOF(q_stEP1908_Diag.wMC1Temp);
			fbCoERead.bExecute	:= 	TRUE;		
			iState := iState + 10;		
			
	90:// Evaluate read Micro Controller (MC1) Temperature in DegC of the EP1908.			
		IF NOT fbCoERead.bBusy THEN
			fbCoERead.bExecute := FALSE;
			q_sErrorDescription := 'No Error';
			iState := iState + 10;
			IF fbCoERead.bError THEN
				q_sErrorDescription := 'EP1908 MC1 Temp - Read Error';
			END_IF
		END_IF	

	100:// Set Parameters to read Micro Controller (MC2) Temperature in DegC of the EP1908.			
			fbCoERead.nSubIndex	:= 	16#02;
			fbCoERead.nIndex	:= 	16#FA80;
			fbCoERead.pDstBuf	:= 	ADR(q_stEP1908_Diag.wMC2Temp);
			fbCoERead.cbBufLen	:= 	SIZEOF(q_stEP1908_Diag.wMC2Temp);
			fbCoERead.bExecute	:= 	TRUE;		
			iState := iState + 10;		
		
	110:// Evaluate read Micro Controller (MC2) Temperature in DegC of the EP1908.			
		IF NOT fbCoERead.bBusy THEN
			fbCoERead.bExecute := FALSE;
			q_sErrorDescription := 'No Error';
			iState := iState + 10;
			IF fbCoERead.bError THEN
				q_sErrorDescription := 'EP1908 MC2 Temp - Read Error';
			END_IF
		END_IF	
		
	120:// Set Parameters to read Micro Controller (MC1) 3300mv Nominal Voltage INPUT of the EP1908.			
			fbCoERead.nSubIndex	:= 	16#01;
			fbCoERead.nIndex	:= 	16#FA81;
			fbCoERead.pDstBuf	:= 	ADR(wEP1908_MC1_3300mV);
			fbCoERead.cbBufLen	:= 	SIZEOF(wEP1908_MC1_3300mV);
			fbCoERead.bExecute	:= 	TRUE;		
			iState := iState + 10;		
		
	130:// Evaluate read Micro Controller (MC1) 3300mv Nominal Voltage INPUT of the EP1908.			
		IF NOT fbCoERead.bBusy THEN
		 	q_stEP1908_Diag.lrMC1_3300mV :=  WORD_TO_LREAL(wEP1908_MC1_3300mV);
			fbCoERead.bExecute := FALSE;
			q_sErrorDescription := 'No Error';
			iState := iState + 10;
			IF fbCoERead.bError THEN
				q_sErrorDescription := 'EP1908 MC1 3.3v Input - Read Error';
			END_IF
		END_IF		
	
	140:// Set Parameters to read Micro Controller (MC2) 3300mv Nominal Voltage INPUT of the EP1908.			
			fbCoERead.nSubIndex	:= 	16#02;
			fbCoERead.nIndex	:= 	16#FA81;
			fbCoERead.pDstBuf	:= 	ADR(wEP1908_MC2_3300mV);
			fbCoERead.cbBufLen	:= 	SIZEOF(wEP1908_MC2_3300mV);
			fbCoERead.bExecute	:= 	TRUE;		
			iState := iState + 10;		
			
	150:// Evaluate read Micro Controller (MC2) 3300mv Nominal Voltage INPUT of the EP1908.			
		IF NOT fbCoERead.bBusy THEN
  			q_stEP1908_Diag.lrMC2_3300mV:=  WORD_TO_LREAL(wEP1908_MC2_3300mV);
			fbCoERead.bExecute := FALSE;
			q_sErrorDescription := 'No Error';
			iState := iState + 10;
			IF fbCoERead.bError THEN
				q_sErrorDescription := 'EP1908 MC2 3.3v Input - Read Error';
			END_IF
		END_IF			
		
	160:// Set Parameters to read Operating Mode of the EP1908.			
			fbCoERead.nSubIndex	:= 	16#01;
			fbCoERead.nIndex	:= 	16#8000;
			fbCoERead.pDstBuf	:= 	ADR(wEP1908_OperMode);
			fbCoERead.cbBufLen	:= 	SIZEOF(wEP1908_OperMode);
			fbCoERead.bExecute	:= 	TRUE;		
			iState := iState + 10;	
			
	170:// Evaluate read Operating Mode of the EP1908.		
		IF NOT fbCoERead.bBusy THEN
  			IF wEP1908_OperMode  =  0 THEN
				q_stEP1908_Diag.sOpMode  :=  'Digital' ;
			ELSIF wEP1908_OperMode  =  1 THEN
				q_stEP1908_Diag.sOpMode  :=  'Standstill Monitoring 1' ;
			ELSIF wEP1908_OperMode  =  2 THEN
				q_stEP1908_Diag.sOpMode  :=  'Standstill Monitoring 2' ;
			ELSE
				q_stEP1908_Diag.sOpMode  :=  'Invalid Mode' ;
			END_IF ;
			fbCoERead.bExecute := FALSE;
			q_sErrorDescription := 'No Error';
			iState := iState + 10;
			IF fbCoERead.bError THEN
				q_sErrorDescription := 'EP1908 Operating Mode - Read Error';
			END_IF
		END_IF		
				
	180:// Set Parameters to read Sensor Test Active/Inactive of the EP1908.			
			fbCoEReadEX.nSubIndex	:= 	1;
			fbCoEReadEX.nIndex	:= 	16#8001;
			fbCoEReadEX.pDstBuf	:= 	ADR(iSensorTestActive);
			fbCoEReadEX.cbBufLen	:= 	SIZEOF(iSensorTestActive);
			fbCoEReadEX.bExecute	:= 	TRUE;		
			iState := iState + 10;	
			
	190:// Evaluate read Sensor Test Active/Inactive of the EP1908.		
		IF NOT fbCoEReadEX.bBusy THEN
  			IF NOT iSensorTestActive.0 THEN
				q_stEP1908_Diag.xSensorTestActive1 := FALSE;	
			ELSIF iSensorTestActive.0 THEN
				q_stEP1908_Diag.xSensorTestActive1 := TRUE;	
			END_IF
				
			IF NOT iSensorTestActive.1 THEN
				q_stEP1908_Diag.xSensorTestActive2 := FALSE;	
			ELSIF iSensorTestActive.1 THEN
				q_stEP1908_Diag.xSensorTestActive2 := TRUE;
			END_IF
				
			IF NOT iSensorTestActive.2 THEN
				q_stEP1908_Diag.xSensorTestActive3 := FALSE;	
			ELSIF iSensorTestActive.2 THEN
				q_stEP1908_Diag.xSensorTestActive3 := TRUE;
			END_IF	
				
			IF NOT iSensorTestActive.3 THEN
				q_stEP1908_Diag.xSensorTestActive4 := FALSE;	
			ELSIF iSensorTestActive.3 THEN
				q_stEP1908_Diag.xSensorTestActive4 := TRUE;
			END_IF
				
			IF NOT iSensorTestActive.4 THEN
				q_stEP1908_Diag.xSensorTestActive5 := FALSE;	
			ELSIF iSensorTestActive.4 THEN
				q_stEP1908_Diag.xSensorTestActive5 := TRUE;	
			END_IF
				
			IF NOT iSensorTestActive.5 THEN
				q_stEP1908_Diag.xSensorTestActive6 := FALSE;	
			ELSIF iSensorTestActive.5 THEN
				q_stEP1908_Diag.xSensorTestActive6 := TRUE;
			END_IF
				
			IF NOT iSensorTestActive.6 THEN
				q_stEP1908_Diag.xSensorTestActive7 := FALSE;	
			ELSIF iSensorTestActive.6 THEN
				q_stEP1908_Diag.xSensorTestActive7 := TRUE;	
			END_IF
				
			IF NOT iSensorTestActive.7 THEN
				q_stEP1908_Diag.xSensorTestActive8 := FALSE;	
			ELSIF iSensorTestActive.7 THEN
				q_stEP1908_Diag.xSensorTestActive8 := TRUE;
			END_IF
			fbCoEReadEX.bExecute := FALSE;
			q_sErrorDescription := 'No Error';
			iState := iState + 10;
			IF fbCoEReadEX.bError THEN
				q_sErrorDescription := 'EP1908 Sensor Test - Read Error';
			END_IF
		END_IF		
			
	200:// Set Parameters to read Logic of Channels 1 and 2 of the EP1908.			
	(* -- SPEED/FREQUENCY MEASUREMENT --
		The permitted frequency range is 2Hz - 50Hz. Values below are reported as 0Hz. Values above result in a 
		diagnostic message which can be reset by the rising edge at the SAFE Output signal ErrAck of the EP1908-0002. *)
			fbCoERead.nSubIndex	:= 	1;
			fbCoERead.nIndex	:= 	16#8002;
			fbCoERead.pDstBuf	:= 	ADR(bEP1908_Logic1_2);
			fbCoERead.cbBufLen	:= 	SIZEOF(bEP1908_Logic1_2);
			fbCoERead.bExecute	:= 	TRUE;		
			iState := iState + 10;	

	210:// Evaluate read Logic of Channels 1 and 2 of the EP1908.		
	(* -- SPEED/FREQUENCY MEASUREMENT --
		The permitted frequency range is 2Hz - 50Hz. Values below are reported as 0Hz. Values above result in a 
		diagnostic message which can be reset by the rising edge at the SAFE Output signal ErrAck of the EP1908-0002. *)
		IF NOT fbCoERead.bBusy THEN
  			IF  bEP1908_Logic1_2  = 0  THEN
				q_stEP1908_Diag.sLogicMode_Ch1Ch2  := 'Single Channel Logic.' ;
			ELSIF  bEP1908_Logic1_2  = 1  THEN
				q_stEP1908_Diag.sLogicMode_Ch1Ch2  := 'Asynchronous Analysis OSSD. Sensor Test Must be Disabled!' ;
			ELSIF  bEP1908_Logic1_2  = 2  THEN
				q_stEP1908_Diag.sLogicMode_Ch1Ch2  := 'Any Pulse Repetition OSSD. Sensor Test Must be Disabled!' ;
			ELSIF  bEP1908_Logic1_2  = 3  THEN
				q_stEP1908_Diag.sLogicMode_Ch1Ch2  := 'Short Cut, No Module Fault. Sensor Test be Enabled!' ;
			ELSIF  bEP1908_Logic1_2  = 4  THEN
				q_stEP1908_Diag.sLogicMode_Ch1Ch2  := 'Velocity Control (1), Single Logic (2).' ;
			ELSIF  bEP1908_Logic1_2  = 5  THEN
				q_stEP1908_Diag.sLogicMode_Ch1Ch2  := 'Single Logic (1), Velocity Control (2).' ;
			ELSIF  bEP1908_Logic1_2  = 6  THEN
				q_stEP1908_Diag.sLogicMode_Ch1Ch2  := 'Velocity Control.' ;
			ELSIF  bEP1908_Logic1_2  = 7  THEN
				q_stEP1908_Diag.sLogicMode_Ch1Ch2  := 'Two Channel Synchronous Velocity Control.' ;
			ELSIF  bEP1908_Logic1_2  = 8  THEN
				q_stEP1908_Diag.sLogicMode_Ch1Ch2  := 'Two Channel Encoder Velocity Control.' ;
			ELSIF  bEP1908_Logic1_2  = 9  THEN
				q_stEP1908_Diag.sLogicMode_Ch1Ch2  := 'Two Channel Asynchronous Veloctiy Control.' ;
			ELSE
				q_stEP1908_Diag.sLogicMode_Ch1Ch2  := 'Invalid Logic CH3 and CH4' ;
			END_IF ;	
			fbCoERead.bExecute := FALSE;
			q_sErrorDescription := 'No Error';
			iState := iState + 10;
			IF fbCoERead.bError THEN
				q_sErrorDescription := 'EP1908 Logic of Channels 1 and 2 - Read Error';
			END_IF
		END_IF		

	220:// Set Parameters to read Logic of Channels 3 and 4 of the EP1908.	
	(* -- SPEED/FREQUENCY MEASUREMENT --
		The permitted frequency range is 2Hz - 50Hz. Values below are reported as 0Hz. Values above result in a 
		diagnostic message which can be reset by the rising edge at the SAFE Output signal ErrAck of the EP1908-0002. *)
			fbCoERead.nSubIndex	:= 	5;
			fbCoERead.nIndex	:= 	16#8002;
			fbCoERead.pDstBuf	:= 	ADR(bEP1908_Logic3_4);
			fbCoERead.cbBufLen	:= 	SIZEOF(bEP1908_Logic3_4);
			fbCoERead.bExecute	:= 	TRUE;		
			iState := iState + 10;	
			
	230:// Evaluate read Logic of Channels 3 and 4 of the EP1908.		
	(* -- SPEED/FREQUENCY MEASUREMENT --
		The permitted frequency range is 2Hz - 50Hz. Values below are reported as 0Hz. Values above result in a 
		diagnostic message which can be reset by the rising edge at the SAFE Output signal ErrAck of the EP1908-0002. *)
		IF NOT fbCoERead.bBusy THEN
  			IF  bEP1908_Logic3_4  = 0  THEN
				q_stEP1908_Diag.sLogicMode_Ch3Ch4  := 'Single Channel Logic.' ;
			ELSIF  bEP1908_Logic3_4  = 1  THEN
				q_stEP1908_Diag.sLogicMode_Ch3Ch4  := 'Asynchronous Analysis OSSD. Sensor Test Must Be OFF!' ;
			ELSIF  bEP1908_Logic3_4  = 2  THEN
				q_stEP1908_Diag.sLogicMode_Ch3Ch4  := 'Any Pulse Repetition OSSD. Sensor Test Must Be OFF!' ;
			ELSIF  bEP1908_Logic3_4  = 3  THEN
				q_stEP1908_Diag.sLogicMode_Ch3Ch4  := 'Short Cut, No Module Fault. Sensor Test Must Be ON!' ;
			ELSIF  bEP1908_Logic3_4  = 4  THEN
				q_stEP1908_Diag.sLogicMode_Ch3Ch4  := 'Velocity Control (3), Single Logic (4).' ;
			ELSIF  bEP1908_Logic3_4  = 5  THEN
				q_stEP1908_Diag.sLogicMode_Ch3Ch4  := 'Single Logic (3), Velocity Control (4).' ;
			ELSIF  bEP1908_Logic3_4  = 6  THEN
				q_stEP1908_Diag.sLogicMode_Ch3Ch4  := 'Velocity Control.' ;
			ELSIF  bEP1908_Logic3_4  = 7  THEN
				q_stEP1908_Diag.sLogicMode_Ch3Ch4  := 'Two Channel Synchronous Velocity Control.' ;
			ELSIF  bEP1908_Logic3_4  = 8  THEN
				q_stEP1908_Diag.sLogicMode_Ch3Ch4  := 'Two Channel Encoder Velocity Control.' ;
			ELSIF  bEP1908_Logic3_4  = 9  THEN
				q_stEP1908_Diag.sLogicMode_Ch3Ch4  := 'Two Channel Asynchronous Veloctiy Control.' ;
			ELSE
				q_stEP1908_Diag.sLogicMode_Ch3Ch4  := 'Invalid Logic CH3 and CH4' ;
			END_IF ;		
			fbCoERead.bExecute := FALSE;
			q_sErrorDescription := 'No Error';
			iState := iState + 10;
			IF fbCoERead.bError THEN
				q_sErrorDescription := 'EP1908 Logic of Channels 3 and 4 - Read Error';
			END_IF
		END_IF			
		
	240:// Set Parameters to read Logic of Channels 5 and 6 of the EP1908.	
	(* -- SPEED/FREQUENCY MEASUREMENT --
		The permitted frequency range is 2Hz - 50Hz. Values below are reported as 0Hz. Values above result in a 
		diagnostic message which can be reset by the rising edge at the SAFE Output signal ErrAck of the EP1908-0002. *)
			fbCoERead.nSubIndex	:= 	9;
			fbCoERead.nIndex	:= 	16#8002;
			fbCoERead.pDstBuf	:= 	ADR(bEP1908_Logic5_6);
			fbCoERead.cbBufLen	:= 	SIZEOF(bEP1908_Logic5_6);
			fbCoERead.bExecute	:= 	TRUE;		
			iState := iState + 10;	
			
	250:// Evaluate read Logic of Channels 5 and 6 of the EP1908.		
	(* -- SPEED/FREQUENCY MEASUREMENT --
		The permitted frequency range is 2Hz - 50Hz. Values below are reported as 0Hz. Values above result in a 
		diagnostic message which can be reset by the rising edge at the SAFE Output signal ErrAck of the EP1908-0002. *)
		IF NOT fbCoERead.bBusy THEN
  			IF  bEP1908_Logic5_6  = 0  THEN
				q_stEP1908_Diag.sLogicMode_Ch5Ch6  := 'Single Channel Logic.' ;
			ELSIF  bEP1908_Logic5_6  =  1  THEN
				q_stEP1908_Diag.sLogicMode_Ch5Ch6  := 'Asynchronous Analysis OSSD. Sensor Test Must Be OFF!' ;
			ELSIF  bEP1908_Logic5_6  =  2  THEN
				q_stEP1908_Diag.sLogicMode_Ch5Ch6  := 'Any Pulse Repetition OSSD. Sensor Test Must Be OFF!' ;
			ELSIF  bEP1908_Logic5_6  =  3  THEN
				q_stEP1908_Diag.sLogicMode_Ch5Ch6  := 'Short Cut, No Module Fault. Sensor Test Must Be ON!' ;
			ELSIF  bEP1908_Logic5_6  =  4  THEN
				q_stEP1908_Diag.sLogicMode_Ch5Ch6  := 'Velocity Control (5), Single Logic (6).' ;
			ELSIF  bEP1908_Logic5_6  =  5  THEN
				q_stEP1908_Diag.sLogicMode_Ch5Ch6  := 'Single Logic (5), Velocity Control (6).' ;
			ELSIF  bEP1908_Logic5_6  =  6  THEN
				q_stEP1908_Diag.sLogicMode_Ch5Ch6  := 'Velocity Control.' ;
			ELSIF  bEP1908_Logic5_6  =  7  THEN
				q_stEP1908_Diag.sLogicMode_Ch5Ch6  := 'Two Channel Synchronous Velocity Control.' ;
			ELSIF  bEP1908_Logic5_6  =  8  THEN
				q_stEP1908_Diag.sLogicMode_Ch5Ch6  := 'Two Channel Encoder Velocity Control.' ;
			ELSIF  bEP1908_Logic5_6  =  9  THEN
				q_stEP1908_Diag.sLogicMode_Ch5Ch6  := 'Two Channel Asynchronous Veloctiy Control.' ;
			ELSE
				q_stEP1908_Diag.sLogicMode_Ch5Ch6 := 'Invalid Logic CH5 and CH6' ;
			END_IF ;			
			fbCoERead.bExecute := FALSE;
			q_sErrorDescription := 'No Error';
			iState := iState + 10;
			IF fbCoERead.bError THEN
				q_sErrorDescription := 'EP1908 Logic of Channels 5 and 6 - Read Error';
			END_IF
		END_IF			
	
	260:// Set Parameters to read Logic of Channels 7 and 8 of the EP1908.	
	(* -- SPEED/FREQUENCY MEASUREMENT --
		The permitted frequency range is 2Hz - 50Hz. Values below are reported as 0Hz. Values above result in a 
		diagnostic message which can be reset by the rising edge at the SAFE Output signal ErrAck of the EP1908-0002. *)
			fbCoERead.nSubIndex	:= 	16#0D;
			fbCoERead.nIndex	:= 	16#8002;
			fbCoERead.pDstBuf	:= 	ADR(bEP1908_Logic7_8);
			fbCoERead.cbBufLen	:= 	SIZEOF(bEP1908_Logic7_8);
			fbCoERead.bExecute	:= 	TRUE;		
			iState := iState + 10;	
			
	270:// Evaluate read Logic of Channels 7 and 8 of the EP1908.		
	(* -- SPEED/FREQUENCY MEASUREMENT --
		The permitted frequency range is 2Hz - 50Hz. Values below are reported as 0Hz. Values above result in a 
		diagnostic message which can be reset by the rising edge at the SAFE Output signal ErrAck of the EP1908-0002. *)
		IF NOT fbCoERead.bBusy THEN
  			IF  bEP1908_Logic7_8  = 0  THEN
				q_stEP1908_Diag.sLogicMode_Ch7Ch8  := 'Single Channel Logic.' ;
			ELSIF  bEP1908_Logic7_8  = 1  THEN
				q_stEP1908_Diag.sLogicMode_Ch7Ch8  := 'Asynchronous Analysis OSSD. Sensor Test Must Be OFF!' ;
			ELSIF  bEP1908_Logic7_8  = 2  THEN
				q_stEP1908_Diag.sLogicMode_Ch7Ch8  := 'Any Pulse Repetition OSSD. Sensor Test Must Be OFF!' ;
			ELSIF  bEP1908_Logic7_8  = 3  THEN
				q_stEP1908_Diag.sLogicMode_Ch7Ch8  := 'Short Cut, No Module Fault. Sensor Test Must Be ON!' ;
			ELSIF  bEP1908_Logic7_8  = 4  THEN
				q_stEP1908_Diag.sLogicMode_Ch7Ch8  := 'Velocity Control (7), Single Logic (8).' ;
			ELSIF  bEP1908_Logic7_8  = 5  THEN
				q_stEP1908_Diag.sLogicMode_Ch7Ch8  := 'Single Logic (7), Velocity Control (8).' ;
			ELSIF  bEP1908_Logic7_8  = 6  THEN
				q_stEP1908_Diag.sLogicMode_Ch7Ch8  := 'Velocity Control.' ;
			ELSIF  bEP1908_Logic7_8  = 7  THEN
				q_stEP1908_Diag.sLogicMode_Ch7Ch8  := 'Two Channel Synchronous Velocity Control.' ;
			ELSIF  bEP1908_Logic7_8  = 8  THEN
				q_stEP1908_Diag.sLogicMode_Ch7Ch8  := 'Two Channel Encoder Velocity Control.' ;
			ELSIF  bEP1908_Logic7_8  = 9  THEN
				q_stEP1908_Diag.sLogicMode_Ch7Ch8  := 'Two Channel Asynchronous Veloctiy Control.' ;
			ELSE
				q_stEP1908_Diag.sLogicMode_Ch7Ch8  := 'Invalid Logic CH7 and CH8' ;
			END_IF ;			
			fbCoERead.bExecute := FALSE;
			q_sErrorDescription := 'No Error';
			iState := iState + 10;
			IF fbCoERead.bError THEN
				q_sErrorDescription := 'EP1908 Logic of Channels 7 and 8 - Read Error';
			END_IF
		END_IF		
		
	280:// Set Parameters to read Velocity/Frequency Limits of the EP1908.	
			fbCoEReadEX.nSubIndex	:= 	1;
			fbCoEReadEX.nIndex		:= 	16#8003;
			fbCoEReadEX.pDstBuf		:= 	ADR(arrEP1908_VelocityLimit);
			fbCoEReadEX.cbBufLen	:= 	SIZEOF(arrEP1908_VelocityLimit);
			fbCoEReadEX.bExecute	:= 	TRUE;		
			iState := iState + 10;	
			
	290:// Evaluate read Velocity/Frequency Limits of the EP1908.			
		IF NOT fbCoEReadEX.bBusy THEN
  			q_stEP1908_Diag.iEP1908_VelocityLimitCh1 := arrEP1908_VelocityLimit[0];
			q_stEP1908_Diag.iEP1908_VelocityLimitCh2 := arrEP1908_VelocityLimit[1];
			q_stEP1908_Diag.iEP1908_VelocityLimitCh3 := arrEP1908_VelocityLimit[2];
			q_stEP1908_Diag.iEP1908_VelocityLimitCh4 := arrEP1908_VelocityLimit[3];
			q_stEP1908_Diag.iEP1908_VelocityLimitCh5 := arrEP1908_VelocityLimit[4];
			q_stEP1908_Diag.iEP1908_VelocityLimitCh6 := arrEP1908_VelocityLimit[5];
			q_stEP1908_Diag.iEP1908_VelocityLimitCh7 := arrEP1908_VelocityLimit[6];
			q_stEP1908_Diag.iEP1908_VelocityLimitCh8 := arrEP1908_VelocityLimit[7];	
			fbCoEReadEX.bExecute := FALSE;
			q_sErrorDescription := 'No Error';
			iState := iState + 10;
			IF fbCoEReadEX.bError THEN
				q_sErrorDescription := 'EP1908 Velocity/Frequency Limits - Read Error';
			END_IF
		END_IF			

	300:// Set Parameters to read Actual Velocity/Frequency  of the EP1908.	
			fbCoEReadEX.nSubIndex	:= 	1;
			fbCoEReadEX.nIndex		:= 	16#A008;
			fbCoEReadEX.pDstBuf		:= 	ADR(arrEP1908ActualVelocities);
			fbCoEReadEX.cbBufLen	:= 	SIZEOF(arrEP1908ActualVelocities);
			fbCoEReadEX.bExecute	:= 	TRUE;		
			iState := iState + 10;	
			
	310:// Evaluate read Actual Velocity/Frequency  of the EP1908.			
		IF NOT fbCoEReadEX.bBusy THEN
  			q_stEP1908_Diag.iEP1908_ActVeloctiyCh1 := arrEP1908ActualVelocities[0];
			q_stEP1908_Diag.iEP1908_ActVeloctiyCh2 := arrEP1908ActualVelocities[1];
			q_stEP1908_Diag.iEP1908_ActVeloctiyCh3 := arrEP1908ActualVelocities[2];
			q_stEP1908_Diag.iEP1908_ActVeloctiyCh4 := arrEP1908ActualVelocities[3];
			q_stEP1908_Diag.iEP1908_ActVeloctiyCh5 := arrEP1908ActualVelocities[4];
			q_stEP1908_Diag.iEP1908_ActVeloctiyCh6 := arrEP1908ActualVelocities[5];
			q_stEP1908_Diag.iEP1908_ActVeloctiyCh7 := arrEP1908ActualVelocities[6];
			q_stEP1908_Diag.iEP1908_ActVeloctiyCh8 := arrEP1908ActualVelocities[7];
			fbCoEReadEX.bExecute := FALSE;
			q_sErrorDescription := 'No Error';
			iState := iState + 10;
			IF fbCoEReadEX.bError THEN
				q_sErrorDescription := 'EP1908 Actual Velocity/Frequency - Read Error';
			END_IF
		END_IF		
	
	320:// Set Parameters to read Max Velocity/Frequency of the EP1908.	
			(* Max value since the last Startup of TwinSAFE. *)
			fbCoEReadEX.nSubIndex	:= 	1;
			fbCoEReadEX.nIndex		:= 	16#A009;
			fbCoEReadEX.pDstBuf		:= 	ADR(arrEP1908MaxVelocities);
			fbCoEReadEX.cbBufLen	:= 	SIZEOF(arrEP1908MaxVelocities);
			fbCoEReadEX.bExecute	:= 	TRUE;		
			iState := iState + 10;	
			
	330:// Evaluate read Max Velocity/Frequency of the EP1908.		
			(* Max value since the last Startup of TwinSAFE. *)	
		IF NOT fbCoEReadEX.bBusy THEN
  			q_stEP1908_Diag.iEP1908_MaxVeloctiyCh1 := arrEP1908MaxVelocities[0];
			q_stEP1908_Diag.iEP1908_MaxVeloctiyCh2 := arrEP1908MaxVelocities[1];
			q_stEP1908_Diag.iEP1908_MaxVeloctiyCh3 := arrEP1908MaxVelocities[2];
			q_stEP1908_Diag.iEP1908_MaxVeloctiyCh4 := arrEP1908MaxVelocities[3];
			q_stEP1908_Diag.iEP1908_MaxVeloctiyCh5 := arrEP1908MaxVelocities[4];
			q_stEP1908_Diag.iEP1908_MaxVeloctiyCh6 := arrEP1908MaxVelocities[5];
			q_stEP1908_Diag.iEP1908_MaxVeloctiyCh7 := arrEP1908MaxVelocities[6];
			q_stEP1908_Diag.iEP1908_MaxVeloctiyCh8 := arrEP1908MaxVelocities[7];
			fbCoEReadEX.bExecute := FALSE;
			q_sErrorDescription := 'No Error';
			iState := iState + 10;
			IF fbCoEReadEX.bError THEN
				q_sErrorDescription := 'EP1908 Max Velocity/Frequency - Read Error';
			END_IF
		END_IF		
	
	
(**************************************ALARMS**************************************)
(**************************************ALARMS**************************************)
(**************************************ALARMS**************************************)
	340:// Set Parameters to read Sensor Test Error of the EP1908.
			fbCoERead.nSubIndex	:= 	16#0A;
			fbCoERead.nIndex	:= 	16#800E;
			fbCoERead.pDstBuf	:= 	ADR(wEP1908_SenT);
			fbCoERead.cbBufLen	:= 	SIZEOF(wEP1908_SenT);
			fbCoERead.bExecute	:= 	TRUE;		
			iState := iState + 10;	
			
	350:// Evaluate read Sensor Test Error of the EP1908.			
		IF NOT fbCoERead.bBusy THEN
  			(*These errors may only be present temporarily so they need to be latched and then cleared
				to be properly noted by the operator. *)
			IF wEP1908_SenT > 0 THEN
				q_stEP1908_Diag.xSensorTest1_Error 	:= 	wEP1908_SenT.0;
				q_stEP1908_Diag.xSensorTest2_Error 	:= 	wEP1908_SenT.1;
				q_stEP1908_Diag.xSensorTest3_Error 	:= 	wEP1908_SenT.2;
				q_stEP1908_Diag.xSensorTest4_Error 	:=  wEP1908_SenT.3;
				q_stEP1908_Diag.xSensorTest5_Error 	:= 	wEP1908_SenT.4;
				q_stEP1908_Diag.xSensorTest6_Error 	:= 	wEP1908_SenT.5;
				q_stEP1908_Diag.xSensorTest7_Error 	:= 	wEP1908_SenT.6;
				q_stEP1908_Diag.xSensorTest8_Error 	:=  wEP1908_SenT.7;
			ELSIF i_xLatchedMessageReset THEN
				q_stEP1908_Diag.xSensorTest1_Error	:= FALSE;
				q_stEP1908_Diag.xSensorTest2_Error	:= FALSE;
				q_stEP1908_Diag.xSensorTest3_Error	:= FALSE;
				q_stEP1908_Diag.xSensorTest4_Error	:= FALSE;
				q_stEP1908_Diag.xSensorTest5_Error	:= FALSE;
				q_stEP1908_Diag.xSensorTest6_Error	:= FALSE;
				q_stEP1908_Diag.xSensorTest7_Error	:= FALSE;
				q_stEP1908_Diag.xSensorTest8_Error	:= FALSE;
			END_IF
			fbCoERead.bExecute := FALSE;
			q_sErrorDescription := 'No Error';
			iState := iState + 10;
			IF fbCoERead.bError THEN
				q_sErrorDescription := 'EP1908 Sensor Test Error - Read Error';
			END_IF
		END_IF		

	360:// Set Parameters to read Error During Two-Channel Evaluation - Diagnostic object 800E:0B of the EP1908.	
		(* The two channels contradict each other (not same value). *)	
			fbCoERead.nSubIndex	:= 	16#0B;
			fbCoERead.nIndex	:= 	16#800E;
			fbCoERead.pDstBuf	:= 	ADR(wEP1908_2CHEval);
			fbCoERead.cbBufLen	:= 	SIZEOF(wEP1908_2CHEval);
			fbCoERead.bExecute	:= 	TRUE;		
			iState := iState + 10;	
			
	370:// Evaluate read Error During Two-Channel Evaluation - Diagnostic object 800E:0B of the EP1908.		
		(* The two channels contradict each other (not same value). *)	
		IF NOT fbCoERead.bBusy THEN
  			(*These errors may only be present temporarily so they need to be latched and then cleared
				to be properly noted by the operator. *)
			IF wEP1908_2CHEval.0 OR wEP1908_2CHEval.1 OR wEP1908_2CHEval.2 OR wEP1908_2CHEval.3 THEN
				q_stEP1908_Diag.x2ChanEvalError_Pair1	 :=  wEP1908_2CHEval.0;
				q_stEP1908_Diag.x2ChanEvalError_Pair2	 :=  wEP1908_2CHEval.1;
				q_stEP1908_Diag.x2ChanEvalError_Pair1	 :=  wEP1908_2CHEval.2;
				q_stEP1908_Diag.x2ChanEvalError_Pair2	 :=  wEP1908_2CHEval.3;
			ELSIF i_xLatchedMessageReset THEN
				q_stEP1908_Diag.x2ChanEvalError_Pair1	:= FALSE;
				q_stEP1908_Diag.x2ChanEvalError_Pair2	:= FALSE;
				q_stEP1908_Diag.x2ChanEvalError_Pair3	:= FALSE;
				q_stEP1908_Diag.x2ChanEvalError_Pair4	:= FALSE;
			END_IF	
			fbCoERead.bExecute := FALSE;
			q_sErrorDescription := 'No Error';
			iState := iState + 10;
			IF fbCoERead.bError THEN
				q_sErrorDescription := 'EP1908 Error During Two-Channel Evaluation - Read Error';
			END_IF
		END_IF		


	380:// Set Parameters to read Error In Safety Mat Operating Mode: Input Pair Disagree - Diagnostic object 800E:0C of the EP1908.	
		(* The two channels contradict each other (not same value). *)	
			fbCoERead.nSubIndex	:= 	16#0C;
			fbCoERead.nIndex	:= 	16#800E;
			fbCoERead.pDstBuf	:= 	ADR(wEP1908_SMiPair);
			fbCoERead.cbBufLen	:= 	SIZEOF(wEP1908_SMiPair);
			fbCoERead.bExecute	:= 	TRUE;		
			iState := iState + 10;	
			
	390:// Evaluate read read Error In Safety Mat Operating Mode: Input Pair Disagree - Diagnostic object 800E:0C of the EP1908.	
		(* The two channels contradict each other (not same value). *)	
		IF NOT fbCoERead.bBusy THEN
  			(*These errors may only be present temporarily so they need to be latched and then cleared
				to be properly noted by the operator. *)
			IF (wEP1908_SMiPair.0 AND wEP1908_SMiPair.1) OR (wEP1908_SMiPair.2 AND wEP1908_SMiPair.3) OR
				(wEP1908_SMiPair.4 AND wEP1908_SMiPair.5) OR (wEP1908_SMiPair.6 AND wEP1908_SMiPair.7) THEN
				q_stEP1908_Diag.xSafeMatError_Pair1	 :=  (wEP1908_SMiPair.0  AND  wEP1908_SMiPair.1);
				q_stEP1908_Diag.xSafeMatError_Pair2	 :=  (wEP1908_SMiPair.2  AND  wEP1908_SMiPair.3);
				q_stEP1908_Diag.xSafeMatError_Pair3	 :=  (wEP1908_SMiPair.4  AND  wEP1908_SMiPair.5);
				q_stEP1908_Diag.xSafeMatError_Pair4	 :=  (wEP1908_SMiPair.6  AND  wEP1908_SMiPair.7);
			ELSIF i_xLatchedMessageReset THEN
				q_stEP1908_Diag.xSafeMatError_Pair1	:= FALSE;
				q_stEP1908_Diag.xSafeMatError_Pair2	:= FALSE;
				q_stEP1908_Diag.xSafeMatError_Pair3	:= FALSE;
				q_stEP1908_Diag.xSafeMatError_Pair4	:= FALSE;
			END_IF
			fbCoERead.bExecute := FALSE;
			q_sErrorDescription := 'No Error';
			iState := iState + 10;
			IF fbCoERead.bError THEN
				q_sErrorDescription := 'EP1908 Error In Safety Mat: Input Pair Disagree - Read Error';
			END_IF
		END_IF		
	
	400:// Set Parameters to read Error In Safety Mat Operating Mode: External Supply (No test pulses) - Diagnostic object 800E:0D of the EP1908.	
		(* External supply detected (Input channel not getting test pulses). *)	
			fbCoERead.nSubIndex	:= 	16#0D;
			fbCoERead.nIndex	:= 	16#800E;
			fbCoERead.pDstBuf	:= 	ADR(wEP1908_SMExtSupply);
			fbCoERead.cbBufLen	:= 	SIZEOF(wEP1908_SMExtSupply);
			fbCoERead.bExecute	:= 	TRUE;		
			iState := iState + 10;	
	
	410:// Evaluate read read Error In Safety Mat Operating Mode: External Supply (No test pulses) - Diagnostic object 800E:0D of the EP1908.	
		(* The two channels contradict each other (not same value). *)	
		IF NOT fbCoERead.bBusy THEN
  			(*These errors may only be present temporarily so they need to be latched and then cleared
				to be properly noted by the operator. *)
			IF wEP1908_SMExtSupply > 0  THEN
				q_stEP1908_Diag.xSafeMatExternalSupplyErrorCh1  := 	wEP1908_SMExtSupply.0;
				q_stEP1908_Diag.xSafeMatExternalSupplyErrorCh2  := 	wEP1908_SMExtSupply.1;
				q_stEP1908_Diag.xSafeMatExternalSupplyErrorCh3  := 	wEP1908_SMExtSupply.2;
				q_stEP1908_Diag.xSafeMatExternalSupplyErrorCh4  := 	wEP1908_SMExtSupply.3;
				q_stEP1908_Diag.xSafeMatExternalSupplyErrorCh5  := 	wEP1908_SMExtSupply.4;
				q_stEP1908_Diag.xSafeMatExternalSupplyErrorCh6  := 	wEP1908_SMExtSupply.5;
				q_stEP1908_Diag.xSafeMatExternalSupplyErrorCh7  := 	wEP1908_SMExtSupply.6;
				q_stEP1908_Diag.xSafeMatExternalSupplyErrorCh8  := 	wEP1908_SMExtSupply.7;
			ELSIF i_xLatchedMessageReset THEN
				q_stEP1908_Diag.xSafeMatExternalSupplyErrorCh1	:= FALSE;
				q_stEP1908_Diag.xSafeMatExternalSupplyErrorCh2	:= FALSE;
				q_stEP1908_Diag.xSafeMatExternalSupplyErrorCh3	:= FALSE;
				q_stEP1908_Diag.xSafeMatExternalSupplyErrorCh4	:= FALSE;
				q_stEP1908_Diag.xSafeMatExternalSupplyErrorCh5	:= FALSE;
				q_stEP1908_Diag.xSafeMatExternalSupplyErrorCh6	:= FALSE;
				q_stEP1908_Diag.xSafeMatExternalSupplyErrorCh7	:= FALSE;
				q_stEP1908_Diag.xSafeMatExternalSupplyErrorCh8	:= FALSE;
			END_IF
			fbCoERead.bExecute := FALSE;
			q_sErrorDescription := 'No Error';
			iState := iState + 10;
			IF fbCoERead.bError THEN
				q_sErrorDescription := 'EP1908 Error In Safety Mat: External Supply - Read Error';
			END_IF
		END_IF					

	420:// Set Parameters to read Speed Monitoring Error: Overspeed of the EP1908.	
		(* Overspeed was detected at the input. *)
			fbCoERead.nSubIndex	:= 	13;
			fbCoERead.nIndex	:= 	16#800E;
			fbCoERead.pDstBuf	:= 	ADR(wEP1908_SpeedMonitor);
			fbCoERead.cbBufLen	:= 	SIZEOF(wEP1908_SpeedMonitor);
			fbCoERead.bExecute	:= 	TRUE;		
			iState := iState + 10;	
	
		
	430:// Evaluate read Speed Monitoring Error: Overspeed of the EP1908.	
		(* Overspeed was detected at the input. *)
		IF NOT fbCoERead.bBusy THEN
  			(*These errors may only be present temporarily so they need to be latched and then cleared
				to be properly noted by the operator. *)
			IF wEP1908_SpeedMonitor > 0  THEN
				q_stEP1908_Diag.xSpeedMonitorErrorCh1  := 	wEP1908_SpeedMonitor.0;
				q_stEP1908_Diag.xSpeedMonitorErrorCh2  := 	wEP1908_SpeedMonitor.1;
				q_stEP1908_Diag.xSpeedMonitorErrorCh3  := 	wEP1908_SpeedMonitor.2;
				q_stEP1908_Diag.xSpeedMonitorErrorCh4  := 	wEP1908_SpeedMonitor.3;
				q_stEP1908_Diag.xSpeedMonitorErrorCh5  := 	wEP1908_SpeedMonitor.4;
				q_stEP1908_Diag.xSpeedMonitorErrorCh6  := 	wEP1908_SpeedMonitor.5;
				q_stEP1908_Diag.xSpeedMonitorErrorCh7  := 	wEP1908_SpeedMonitor.6;
				q_stEP1908_Diag.xSpeedMonitorErrorCh8  := 	wEP1908_SpeedMonitor.7;
			ELSIF i_xLatchedMessageReset THEN
				q_stEP1908_Diag.xSpeedMonitorErrorCh1	:= FALSE;
				q_stEP1908_Diag.xSpeedMonitorErrorCh2	:= FALSE;
				q_stEP1908_Diag.xSpeedMonitorErrorCh3	:= FALSE;
				q_stEP1908_Diag.xSpeedMonitorErrorCh4	:= FALSE;
				q_stEP1908_Diag.xSpeedMonitorErrorCh5	:= FALSE;
				q_stEP1908_Diag.xSpeedMonitorErrorCh6	:= FALSE;
				q_stEP1908_Diag.xSpeedMonitorErrorCh7	:= FALSE;
				q_stEP1908_Diag.xSpeedMonitorErrorCh8	:= FALSE;
			END_IF
			fbCoERead.bExecute := FALSE;
			q_sErrorDescription := 'No Error';
			iState := iState + 10;
			IF fbCoERead.bError THEN
				q_sErrorDescription := 'EP1908 Speed Monitoring Error: Overspeed - Read Error';
			END_IF
		END_IF				
				
	440:// Set Parameters to read Two Channel Sync Velocity Control Error of the EP1908. 
		(* Both inputs of an input pair were read with inactive State *)
			fbCoERead.nSubIndex	:= 	14;
			fbCoERead.nIndex	:= 	16#800E;
			fbCoERead.pDstBuf	:= 	ADR(wEP1908_2ChSyncVelo);
			fbCoERead.cbBufLen	:= 	SIZEOF(wEP1908_2ChSyncVelo);
			fbCoERead.bExecute	:= 	TRUE;		
			iState := iState + 10;	
		
	450:// Evaluate read Two Channel Sync Velocity Control Error of the EP1908. 
		(* Both inputs of an input pair were read with inactive State *)
		IF NOT fbCoERead.bBusy THEN
  			(*These errors may only be present temporarily so they need to be latched and then cleared
				to be properly noted by the operator. *)
			IF wEP1908_2ChSyncVelo > 0  THEN
				q_stEP1908_Diag.x2ChSyncVelocityErrorPair1  := 	wEP1908_2ChSyncVelo.0;
				q_stEP1908_Diag.x2ChSyncVelocityErrorPair2  := 	wEP1908_2ChSyncVelo.1;
				q_stEP1908_Diag.x2ChSyncVelocityErrorPair3  := 	wEP1908_2ChSyncVelo.2;
				q_stEP1908_Diag.x2ChSyncVelocityErrorPair4  := 	wEP1908_2ChSyncVelo.3;
			ELSIF i_xLatchedMessageReset THEN
				q_stEP1908_Diag.x2ChSyncVelocityErrorPair1	:= FALSE;
				q_stEP1908_Diag.x2ChSyncVelocityErrorPair2	:= FALSE;
				q_stEP1908_Diag.x2ChSyncVelocityErrorPair3	:= FALSE;
				q_stEP1908_Diag.x2ChSyncVelocityErrorPair4	:= FALSE;
			END_IF
			fbCoERead.bExecute := FALSE;
			q_sErrorDescription := 'No Error';
			iState := iState + 10;
			IF fbCoERead.bError THEN
				q_sErrorDescription := 'EP1908 Two Channel Sync Velocity Control Error - Read Error';
			END_IF
		END_IF		
	
	460:// Set Parameters to read Two Channel Sync Velocity Control AND Two Channel Encoder Velocity Control Error of the EP1908. 
		(* Different speeds were identified for the two inputs of an input pair. *)
			fbCoERead.nSubIndex	:= 	15;
			fbCoERead.nIndex	:= 	16#800E;
			fbCoERead.pDstBuf	:= 	ADR(wEP1908_2ChSyncVeloAnd2ChEncVelo);
			fbCoERead.cbBufLen	:= 	SIZEOF(wEP1908_2ChSyncVeloAnd2ChEncVelo);
			fbCoERead.bExecute	:= 	TRUE;		
			iState := iState + 10;	
					
	470:// Evaluate read Two Channel Sync Velocity Control AND Two Channel Encoder Velocity Control Error of the EP1908. 
		(* Different speeds were identified for the two inputs of an input pair. *)
		IF NOT fbCoERead.bBusy THEN
  			(*These errors may only be present temporarily so they need to be latched and then cleared
				to be properly noted by the operator. *)
			IF wEP1908_2ChSyncVeloAnd2ChEncVelo > 0  THEN
				q_stEP1908_Diag.x2ChSyncVeloAnd2ChEncVeloErrorPair1  := 	wEP1908_2ChSyncVeloAnd2ChEncVelo.0;
				q_stEP1908_Diag.x2ChSyncVeloAnd2ChEncVeloErrorPair2  := 	wEP1908_2ChSyncVeloAnd2ChEncVelo.1;
				q_stEP1908_Diag.x2ChSyncVeloAnd2ChEncVeloErrorPair3  := 	wEP1908_2ChSyncVeloAnd2ChEncVelo.2;
				q_stEP1908_Diag.x2ChSyncVeloAnd2ChEncVeloErrorPair4  := 	wEP1908_2ChSyncVeloAnd2ChEncVelo.3;
			ELSIF i_xLatchedMessageReset THEN
				q_stEP1908_Diag.x2ChSyncVeloAnd2ChEncVeloErrorPair1	:= FALSE;
				q_stEP1908_Diag.x2ChSyncVeloAnd2ChEncVeloErrorPair2	:= FALSE;
				q_stEP1908_Diag.x2ChSyncVeloAnd2ChEncVeloErrorPair3	:= FALSE;
				q_stEP1908_Diag.x2ChSyncVeloAnd2ChEncVeloErrorPair4	:= FALSE;
			END_IF
			fbCoERead.bExecute := FALSE;
			q_sErrorDescription := 'No Error';
			iState := iState + 10;
			IF fbCoERead.bError THEN
				q_sErrorDescription := 'EP1908 2 Ch Sync Velocity and 2 Ch Encoder Velocity Error - Read Error';
			END_IF
		END_IF		
	
	480:// Set Parameters to read Connection State of the EP1908.
			fbCoERead.nSubIndex	:= 	1;
			fbCoERead.nIndex	:= 	16#A000;
			fbCoERead.pDstBuf	:= 	ADR(iEP1908_ConnectionState);
			fbCoERead.cbBufLen	:= 	SIZEOF(iEP1908_ConnectionState);
			fbCoERead.bExecute	:= 	TRUE;		
			iState := iState + 10;				
	
	490:// Evaluate read Connection State of the EP1908.
		IF NOT fbCoERead.bBusy THEN
  			IF iEP1908_ConnectionState = 100 THEN
				q_stEP1908_Diag.sConnectionState := 'Reset State';
			ELSIF iEP1908_ConnectionState = 101 THEN
				q_stEP1908_Diag.sConnectionState := 'Session State';
			ELSIF iEP1908_ConnectionState = 102 THEN
				q_stEP1908_Diag.sConnectionState := 'Connection State';
			ELSIF iEP1908_ConnectionState = 103 THEN
				q_stEP1908_Diag.sConnectionState := 'Parameter State';
			ELSIF iEP1908_ConnectionState = 104 THEN
				q_stEP1908_Diag.sConnectionState := 'Data State';
			ELSIF iEP1908_ConnectionState = 105 THEN
				q_stEP1908_Diag.sConnectionState := 'Failsafe State';
			ELSE
				q_stEP1908_Diag.sConnectionState := 'Undefined State';
			END_IF
			fbCoERead.bExecute := FALSE;
			q_sErrorDescription := 'No Error';
			iState := 0;
			IF fbCoERead.bError THEN
				q_sErrorDescription := 'EP1908 Connection State - Read Error';
			END_IF
		END_IF			
END_CASE

// FB_EcCoESdoRead for all CoE reads.
fbCoERead(
	sNetId:= i_sNetId, 
	nSlaveAddr:= i_nSlaveAddr, 
	nSubIndex:= , 
	nIndex:= , 
	pDstBuf:= , 
	cbBufLen:= , 
	bExecute:= , 
	tTimeout:= T#2S, 
	bBusy=> , 
	bError=> q_xError, 
	nErrId=> q_nErrorID);

// FB_EcCoESdoReadEx for all CoE EX reads.
fbCoEReadEX(
	sNetId:= i_sNetId, 
	nSlaveAddr:= i_nSlaveAddr, 
	nSubIndex:= , 
	nIndex:= , 
	pDstBuf:= , 
	cbBufLen:= , 
	bExecute:= , 
	tTimeout:= T#2S, 
	bCompleteAccess:= TRUE, 
	bBusy=> , 
	bError=> q_xError, 
	nErrId=> q_nErrorID);

// If any of above errors exist set q_stEP1908_Diag.xEP1908Error TRUE
IF  NOT q_stEP1908_Diag.x2ChanEvalError_Pair1 OR
	q_stEP1908_Diag.x2ChanEvalError_Pair2 OR
	q_stEP1908_Diag.x2ChanEvalError_Pair3 OR
	q_stEP1908_Diag.x2ChanEvalError_Pair4 OR
	q_stEP1908_Diag.x2ChSyncVeloAnd2ChEncVeloErrorPair1 OR
	q_stEP1908_Diag.x2ChSyncVeloAnd2ChEncVeloErrorPair2 OR
	q_stEP1908_Diag.x2ChSyncVeloAnd2ChEncVeloErrorPair3 OR
	q_stEP1908_Diag.x2ChSyncVeloAnd2ChEncVeloErrorPair4 OR
	q_stEP1908_Diag.x2ChSyncVelocityErrorPair1 OR
	q_stEP1908_Diag.x2ChSyncVelocityErrorPair2 OR
	q_stEP1908_Diag.x2ChSyncVelocityErrorPair3 OR
	q_stEP1908_Diag.x2ChSyncVelocityErrorPair4 OR
	q_stEP1908_Diag.xSafeMatExternalSupplyErrorCh1 OR
	q_stEP1908_Diag.xSafeMatExternalSupplyErrorCh2 OR
	q_stEP1908_Diag.xSafeMatExternalSupplyErrorCh3 OR
	q_stEP1908_Diag.xSafeMatExternalSupplyErrorCh4 OR
	q_stEP1908_Diag.xSafeMatExternalSupplyErrorCh5 OR
	q_stEP1908_Diag.xSafeMatExternalSupplyErrorCh6 OR
	q_stEP1908_Diag.xSafeMatExternalSupplyErrorCh7 OR
	q_stEP1908_Diag.xSafeMatExternalSupplyErrorCh8 OR
	q_stEP1908_Diag.xSensorTest1_Error OR
	q_stEP1908_Diag.xSensorTest2_Error OR
	q_stEP1908_Diag.xSensorTest3_Error OR
	q_stEP1908_Diag.xSensorTest4_Error OR
	q_stEP1908_Diag.xSensorTest5_Error OR
	q_stEP1908_Diag.xSensorTest6_Error OR
	q_stEP1908_Diag.xSensorTest7_Error OR
	q_stEP1908_Diag.xSensorTest8_Error OR
	q_stEP1908_Diag.xSpeedMonitorErrorCh1 OR
	q_stEP1908_Diag.xSpeedMonitorErrorCh2 OR
	q_stEP1908_Diag.xSpeedMonitorErrorCh3 OR
	q_stEP1908_Diag.xSpeedMonitorErrorCh4 OR
	q_stEP1908_Diag.xSpeedMonitorErrorCh5 OR
	q_stEP1908_Diag.xSpeedMonitorErrorCh6 OR
	q_stEP1908_Diag.xSpeedMonitorErrorCh7 OR
	q_stEP1908_Diag.xSpeedMonitorErrorCh8 THEN
		q_stEP1908_Diag.xEP1908Error := FALSE;
ELSIF q_stEP1908_Diag.x2ChanEvalError_Pair1 OR
	q_stEP1908_Diag.x2ChanEvalError_Pair2 OR
	q_stEP1908_Diag.x2ChanEvalError_Pair3 OR
	q_stEP1908_Diag.x2ChanEvalError_Pair4 OR
	q_stEP1908_Diag.x2ChSyncVeloAnd2ChEncVeloErrorPair1 OR
	q_stEP1908_Diag.x2ChSyncVeloAnd2ChEncVeloErrorPair2 OR
	q_stEP1908_Diag.x2ChSyncVeloAnd2ChEncVeloErrorPair3 OR
	q_stEP1908_Diag.x2ChSyncVeloAnd2ChEncVeloErrorPair4 OR
	q_stEP1908_Diag.x2ChSyncVelocityErrorPair1 OR
	q_stEP1908_Diag.x2ChSyncVelocityErrorPair2 OR
	q_stEP1908_Diag.x2ChSyncVelocityErrorPair3 OR
	q_stEP1908_Diag.x2ChSyncVelocityErrorPair4 OR
	q_stEP1908_Diag.xSafeMatExternalSupplyErrorCh1 OR
	q_stEP1908_Diag.xSafeMatExternalSupplyErrorCh2 OR
	q_stEP1908_Diag.xSafeMatExternalSupplyErrorCh3 OR
	q_stEP1908_Diag.xSafeMatExternalSupplyErrorCh4 OR
	q_stEP1908_Diag.xSafeMatExternalSupplyErrorCh5 OR
	q_stEP1908_Diag.xSafeMatExternalSupplyErrorCh6 OR
	q_stEP1908_Diag.xSafeMatExternalSupplyErrorCh7 OR
	q_stEP1908_Diag.xSafeMatExternalSupplyErrorCh8 OR
	q_stEP1908_Diag.xSensorTest1_Error OR
	q_stEP1908_Diag.xSensorTest2_Error OR
	q_stEP1908_Diag.xSensorTest3_Error OR
	q_stEP1908_Diag.xSensorTest4_Error OR
	q_stEP1908_Diag.xSensorTest5_Error OR
	q_stEP1908_Diag.xSensorTest6_Error OR
	q_stEP1908_Diag.xSensorTest7_Error OR
	q_stEP1908_Diag.xSensorTest8_Error OR
	q_stEP1908_Diag.xSpeedMonitorErrorCh1 OR
	q_stEP1908_Diag.xSpeedMonitorErrorCh2 OR
	q_stEP1908_Diag.xSpeedMonitorErrorCh3 OR
	q_stEP1908_Diag.xSpeedMonitorErrorCh4 OR
	q_stEP1908_Diag.xSpeedMonitorErrorCh5 OR
	q_stEP1908_Diag.xSpeedMonitorErrorCh6 OR
	q_stEP1908_Diag.xSpeedMonitorErrorCh7 OR
	q_stEP1908_Diag.xSpeedMonitorErrorCh8 THEN
		q_stEP1908_Diag.xEP1908Error := TRUE;
END_IF

END_FUNCTION_BLOCK
